LIN {X 0,Y 538.019,Z 685.461,A -85,B 0,C 180,E1 -4168.934,E2 -4168.934} C_VEL
LIN {X 0,Y 538.004,Z 685.465,A -85,B 0,C 180,E1 -4171.889,E2 -4171.889} C_VEL
LIN {X 0,Y 538.017,Z 685.462,A -85,B 0,C 180,E1 -4174.621,E2 -4174.621} C_VEL
LIN {X 0,Y 537.998,Z 685.467,A -85,B 0,C 180,E1 -4177.171,E2 -4177.171} C_VEL
LIN {X 0,Y 538.01,Z 685.465,A -85,B 0,C 180,E1 -4180.276,E2 -4180.276} C_VEL
LIN {X 0,Y 537.361,Z 685.545,A -85,B 0,C 180,E1 -4180.901,E2 -4180.901} C_VEL
LIN {X 0,Y 534.509,Z 685.908,A -85,B 0,C 180,E1 -4181.916,E2 -4181.916} C_VEL
LIN {X 0,Y 532.082,Z 686.21,A -85,B 0,C 180,E1 -4182.733,E2 -4182.733} C_VEL
LIN {X 0,Y 531.033,Z 686.336,A -85,B 0,C 180,E1 -4183.364,E2 -4183.364} C_VEL
LIN {X 0,Y 530.945,Z 686.346,A -85,B 0,C 180,E1 -4183.578,E2 -4183.578} C_VEL
LIN {X 0,Y 530.938,Z 686.345,A -85,B 0,C 180,E1 -4186.505,E2 -4186.505} C_VEL
LIN {X 0,Y 530.976,Z 686.345,A -85,B 0,C 180,E1 -4189.568,E2 -4189.568} C_VEL
LIN {X 0,Y 531.016,Z 686.543,A -85,B 0,C 180,E1 -4190.371,E2 -4190.371} C_VEL
LIN {X 0,Y 531.273,Z 687.633,A -85,B 0,C 180,E1 -4190.492,E2 -4190.492} C_VEL
LIN {X 0,Y 532.785,Z 692.095,A -85,B 0,C 180,E1 -4190.606,E2 -4190.606} C_VEL
LIN {X 0,Y 532.506,Z 766.443,A -85,B 0,C 180,E1 -4191.64,E2 -4191.64} C_VEL
LIN {X 0,Y 532.44,Z 779.405,A -85,B 0,C 180,E1 -4191.978,E2 -4191.978} C_VEL
LIN {X 0,Y 532.245,Z 791.35,A -85,B 0,C 180,E1 -4192.434,E2 -4192.434} C_VEL
LIN {X 0,Y 532.057,Z 803.366,A -85,B 0,C 180,E1 -4193.059,E2 -4193.059} C_VEL
LIN {X 0,Y 531.84,Z 814.43,A -85,B 0,C 180,E1 -4193.804,E2 -4193.804} C_VEL
LIN {X 0,Y 531.584,Z 824.165,A -85,B 0,C 180,E1 -4194.617,E2 -4194.617} C_VEL
LIN {X 0,Y 531.338,Z 833.433,A -85,B 0,C 180,E1 -4195.568,E2 -4195.568} C_VEL
LIN {X 0,Y 531.062,Z 842.493,A -85,B 0,C 180,E1 -4196.728,E2 -4196.728} C_VEL
LIN {X 0,Y 530.923,Z 849.848,A -85,B 0,C 180,E1 -4197.908,E2 -4197.908} C_VEL
LIN {X 0,Y 530.783,Z 856.177,A -85,B 0,C 180,E1 -4199.198,E2 -4199.198} C_VEL
LIN {X 0,Y 530.683,Z 860.138,A -85,B 0,C 180,E1 -4200.225,E2 -4200.225} C_VEL
LIN {X 0,Y 530.626,Z 863.895,A -85,B 0,C 180,E1 -4201.524,E2 -4201.524} C_VEL
LIN {X 0,Y 530.54,Z 866.036,A -85,B 0,C 180,E1 -4202.567,E2 -4202.567} C_VEL
LIN {X 0,Y 530.541,Z 866.991,A -85,B 0,C 180,E1 -4203.233,E2 -4203.233} C_VEL
LIN {X 0,Y 530.53,Z 867.86,A -85,B 0,C 180,E1 -4204.265,E2 -4204.265} C_VEL
LIN {X 0,Y 530.494,Z 867.898,A -85,B 0,C 180,E1 -4205.753,E2 -4205.753} C_VEL
LIN {X 0,Y 530.511,Z 867.253,A -85,B 0,C 180,E1 -4206.584,E2 -4206.584} C_VEL
LIN {X 0,Y 530.537,Z 865.086,A -85,B 0,C 180,E1 -4208.017,E2 -4208.017} C_VEL
LIN {X 0,Y 530.666,Z 861.391,A -85,B 0,C 180,E1 -4209.455,E2 -4209.455} C_VEL
LIN {X 0,Y 530.748,Z 857.026,A -85,B 0,C 180,E1 -4210.669,E2 -4210.669} C_VEL
LIN {X 0,Y 530.884,Z 851.4,A -85,B 0,C 180,E1 -4211.876,E2 -4211.876} C_VEL
LIN {X 0,Y 531.012,Z 844.363,A -85,B 0,C 180,E1 -4213.073,E2 -4213.073} C_VEL
LIN {X 0,Y 531.225,Z 837.108,A -85,B 0,C 180,E1 -4214.068,E2 -4214.068} C_VEL
LIN {X 0,Y 531.418,Z 828.24,A -85,B 0,C 180,E1 -4215.064,E2 -4215.064} C_VEL
LIN {X 0,Y 531.703,Z 817.426,A -85,B 0,C 180,E1 -4216.042,E2 -4216.042} C_VEL
LIN {X 0,Y 531.959,Z 806.49,A -85,B 0,C 180,E1 -4216.828,E2 -4216.828} C_VEL
LIN {X 0,Y 532.173,Z 795.377,A -85,B 0,C 180,E1 -4217.454,E2 -4217.454} C_VEL
LIN {X 0,Y 532.331,Z 783.475,A -85,B 0,C 180,E1 -4217.966,E2 -4217.966} C_VEL
LIN {X 0,Y 532.499,Z 770.64,A -85,B 0,C 180,E1 -4218.354,E2 -4218.354} C_VEL
LIN {X 0,Y 532.584,Z 756.116,A -85,B 0,C 180,E1 -4218.609,E2 -4218.609} C_VEL
LIN {X 0,Y 532.658,Z 691.597,A -85,B 0,C 180,E1 -4219.49,E2 -4219.49} C_VEL
LIN {X 0,Y 531.166,Z 687.265,A -85,B 0,C 180,E1 -4219.615,E2 -4219.615} C_VEL
LIN {X 0,Y 530.995,Z 686.43,A -85,B 0,C 180,E1 -4219.757,E2 -4219.757} C_VEL
LIN {X 0,Y 531.004,Z 686.341,A -85,B 0,C 180,E1 -4222.396,E2 -4222.396} C_VEL
LIN {X 0,Y 531.086,Z 686.328,A -85,B 0,C 180,E1 -4224.686,E2 -4224.686} C_VEL
LIN {X 0,Y 531.135,Z 686.324,A -85,B 0,C 180,E1 -4227.726,E2 -4227.726} C_VEL
LIN {X 0,Y 531.131,Z 686.327,A -85,B 0,C 180,E1 -4230.001,E2 -4230.001} C_VEL
LIN {X 0,Y 531.134,Z 686.327,A -85,B 0,C 180,E1 -4232.276,E2 -4232.276} C_VEL
LIN {X 0,Y 531.086,Z 686.326,A -85,B 0,C 180,E1 -4235.316,E2 -4235.316} C_VEL
LIN {X 0,Y 530.985,Z 686.344,A -85,B 0,C 180,E1 -4238.373,E2 -4238.373} C_VEL
LIN {X 0,Y 531.015,Z 686.333,A -85,B 0,C 180,E1 -4241.65,E2 -4241.65} C_VEL
LIN {X 0,Y 531.027,Z 686.337,A -85,B 0,C 180,E1 -4244.952,E2 -4244.952} C_VEL
LIN {X 0,Y 530.977,Z 686.338,A -85,B 0,C 180,E1 -4247.725,E2 -4247.725} C_VEL
LIN {X 0,Y 530.984,Z 686.344,A -85,B 0,C 180,E1 -4250.94,E2 -4250.94} C_VEL
LIN {X 0,Y 530.958,Z 686.341,A -85,B 0,C 180,E1 -4254.031,E2 -4254.031} C_VEL
LIN {X 0,Y 530.943,Z 686.343,A -85,B 0,C 180,E1 -4256.748,E2 -4256.748} C_VEL
LIN {X 0,Y 530.919,Z 686.353,A -85,B 0,C 180,E1 -4259.327,E2 -4259.327} C_VEL
LIN {X 0,Y 530.955,Z 686.34,A -85,B 0,C 180,E1 -4262.098,E2 -4262.098} C_VEL
LIN {X 0,Y 530.953,Z 686.338,A -85,B 0,C 180,E1 -4264.848,E2 -4264.848} C_VEL
LIN {X 0,Y 530.91,Z 686.354,A -85,B 0,C 180,E1 -4267.513,E2 -4267.513} C_VEL
LIN {X 0,Y 530.91,Z 686.346,A -85,B 0,C 180,E1 -4270.441,E2 -4270.441} C_VEL
LIN {X 0,Y 530.922,Z 686.354,A -85,B 0,C 180,E1 -4273.5,E2 -4273.5} C_VEL
LIN {X 0,Y 530.965,Z 686.35,A -85,B 0,C 180,E1 -4275.625,E2 -4275.625} C_VEL
LIN {X 0,Y 530.912,Z 686.347,A -85,B 0,C 180,E1 -4278.556,E2 -4278.556} C_VEL
LIN {X 0,Y 530.918,Z 686.351,A -85,B 0,C 180,E1 -4281.526,E2 -4281.526} C_VEL
LIN {X 0,Y 530.923,Z 686.349,A -85,B 0,C 180,E1 -4284.377,E2 -4284.377} C_VEL
LIN {X 0,Y 530.95,Z 686.343,A -85,B 0,C 180,E1 -4287.132,E2 -4287.132} C_VEL
LIN {X 0,Y 530.937,Z 686.352,A -85,B 0,C 180,E1 -4289.801,E2 -4289.801} C_VEL
LIN {X 0,Y 530.951,Z 686.525,A -85,B 0,C 180,E1 -4292.419,E2 -4292.419} C_VEL
LIN {X 0,Y 531.176,Z 687.511,A -85,B 0,C 180,E1 -4292.538,E2 -4292.538} C_VEL
LIN {X 0,Y 532.707,Z 692.815,A -85,B 0,C 180,E1 -4292.665,E2 -4292.665} C_VEL
LIN {X 0,Y 532.428,Z 761.148,A -85,B 0,C 180,E1 -4293.605,E2 -4293.605} C_VEL
LIN {X 0,Y 532.252,Z 773.625,A -85,B 0,C 180,E1 -4293.908,E2 -4293.908} C_VEL
LIN {X 0,Y 532.095,Z 783.825,A -85,B 0,C 180,E1 -4294.264,E2 -4294.264} C_VEL
LIN {X 0,Y 531.898,Z 792.983,A -85,B 0,C 180,E1 -4294.673,E2 -4294.673} C_VEL
LIN {X 0,Y 531.647,Z 803.731,A -85,B 0,C 180,E1 -4295.288,E2 -4295.288} C_VEL
LIN {X 0,Y 531.438,Z 813.803,A -85,B 0,C 180,E1 -4296.005,E2 -4296.005} C_VEL
LIN {X 0,Y 531.189,Z 822.13,A -85,B 0,C 180,E1 -4296.717,E2 -4296.717} C_VEL
LIN {X 0,Y 531.027,Z 830.575,A -85,B 0,C 180,E1 -4297.586,E2 -4297.586} C_VEL
LIN {X 0,Y 530.865,Z 837.62,A -85,B 0,C 180,E1 -4298.446,E2 -4298.446} C_VEL
LIN {X 0,Y 530.677,Z 844.505,A -85,B 0,C 180,E1 -4299.454,E2 -4299.454} C_VEL
LIN {X 0,Y 530.615,Z 849.821,A -85,B 0,C 180,E1 -4300.386,E2 -4300.386} C_VEL
LIN {X 0,Y 530.529,Z 854.839,A -85,B 0,C 180,E1 -4301.462,E2 -4301.462} C_VEL
LIN {X 0,Y 530.466,Z 858.836,A -85,B 0,C 180,E1 -4302.539,E2 -4302.539} C_VEL
LIN {X 0,Y 530.435,Z 861.509,A -85,B 0,C 180,E1 -4303.449,E2 -4303.449} C_VEL
LIN {X 0,Y 530.334,Z 863.99,A -85,B 0,C 180,E1 -4304.63,E2 -4304.63} C_VEL
LIN {X 0,Y 530.396,Z 865.686,A -85,B 0,C 180,E1 -4306.201,E2 -4306.201} C_VEL
LIN {X 0,Y 530.368,Z 865.993,A -85,B 0,C 180,E1 -4306.981,E2 -4306.981} C_VEL
LIN {X 0,Y 530.454,Z 865.042,A -85,B 0,C 180,E1 -4308.649,E2 -4308.649} C_VEL
LIN {X 0,Y 530.418,Z 864.223,A -85,B 0,C 180,E1 -4309.31,E2 -4309.31} C_VEL
LIN {X 0,Y 530.427,Z 860.91,A -85,B 0,C 180,E1 -4310.851,E2 -4310.851} C_VEL
LIN {X 0,Y 530.496,Z 857.268,A -85,B 0,C 180,E1 -4312.004,E2 -4312.004} C_VEL
LIN {X 0,Y 530.576,Z 852.512,A -85,B 0,C 180,E1 -4313.153,E2 -4313.153} C_VEL
LIN {X 0,Y 530.679,Z 847.651,A -85,B 0,C 180,E1 -4314.109,E2 -4314.109} C_VEL
LIN {X 0,Y 530.723,Z 841.822,A -85,B 0,C 180,E1 -4315.062,E2 -4315.062} C_VEL
LIN {X 0,Y 530.874,Z 834.803,A -85,B 0,C 180,E1 -4316.014,E2 -4316.014} C_VEL
LIN {X 0,Y 531.069,Z 826.32,A -85,B 0,C 180,E1 -4316.966,E2 -4316.966} C_VEL
LIN {X 0,Y 531.336,Z 817.064,A -85,B 0,C 180,E1 -4317.821,E2 -4317.821} C_VEL
LIN {X 0,Y 531.506,Z 808.475,A -85,B 0,C 180,E1 -4318.484,E2 -4318.484} C_VEL
LIN {X 0,Y 531.713,Z 799.665,A -85,B 0,C 180,E1 -4319.053,E2 -4319.053} C_VEL
LIN {X 0,Y 532.003,Z 788.626,A -85,B 0,C 180,E1 -4319.621,E2 -4319.621} C_VEL
LIN {X 0,Y 532.173,Z 777.264,A -85,B 0,C 180,E1 -4320.071,E2 -4320.071} C_VEL
LIN {X 0,Y 532.334,Z 766.23,A -85,B 0,C 180,E1 -4320.378,E2 -4320.378} C_VEL
LIN {X 0,Y 532.483,Z 752.801,A -85,B 0,C 180,E1 -4320.614,E2 -4320.614} C_VEL
LIN {X 0,Y 532.664,Z 691.69,A -85,B 0,C 180,E1 -4321.441,E2 -4321.441} C_VEL
LIN {X 0,Y 531.212,Z 687.28,A -85,B 0,C 180,E1 -4321.564,E2 -4321.564} C_VEL
LIN {X 0,Y 531.068,Z 686.399,A -85,B 0,C 180,E1 -4321.706,E2 -4321.706} C_VEL
LIN {X 0,Y 530.957,Z 686.35,A -85,B 0,C 180,E1 -4323.795,E2 -4323.795} C_VEL
LIN {X 0,Y 531.073,Z 686.336,A -85,B 0,C 180,E1 -4326.077,E2 -4326.077} C_VEL
LIN {X 0,Y 531.021,Z 686.335,A -85,B 0,C 180,E1 -4329.138,E2 -4329.138} C_VEL
LIN {X 0,Y 531.056,Z 686.332,A -85,B 0,C 180,E1 -4331.67,E2 -4331.67} C_VEL
LIN {X 0,Y 531.038,Z 686.333,A -85,B 0,C 180,E1 -4334.955,E2 -4334.955} C_VEL
LIN {X 0,Y 530.988,Z 686.339,A -85,B 0,C 180,E1 -4337.723,E2 -4337.723} C_VEL
LIN {X 0,Y 531.032,Z 686.337,A -85,B 0,C 180,E1 -4340.127,E2 -4340.127} C_VEL
LIN {X 0,Y 530.951,Z 686.351,A -85,B 0,C 180,E1 -4342.573,E2 -4342.573} C_VEL
LIN {X 0,Y 531.005,Z 686.34,A -85,B 0,C 180,E1 -4345.058,E2 -4345.058} C_VEL
LIN {X 0,Y 530.977,Z 686.34,A -85,B 0,C 180,E1 -4347.598,E2 -4347.598} C_VEL
LIN {X 0,Y 530.975,Z 686.341,A -85,B 0,C 180,E1 -4350.197,E2 -4350.197} C_VEL
LIN {X 0,Y 530.973,Z 686.348,A -85,B 0,C 180,E1 -4352.866,E2 -4352.866} C_VEL
LIN {X 0,Y 530.96,Z 686.343,A -85,B 0,C 180,E1 -4355.62,E2 -4355.62} C_VEL
LIN {X 0,Y 530.971,Z 686.343,A -85,B 0,C 180,E1 -4358.653,E2 -4358.653} C_VEL
LIN {X 0,Y 530.999,Z 686.343,A -85,B 0,C 180,E1 -4361.435,E2 -4361.435} C_VEL
LIN {X 0,Y 530.979,Z 686.34,A -85,B 0,C 180,E1 -4364.548,E2 -4364.548} C_VEL
LIN {X 0,Y 530.988,Z 686.341,A -85,B 0,C 180,E1 -4367.834,E2 -4367.834} C_VEL
LIN {X 0,Y 530.976,Z 686.339,A -85,B 0,C 180,E1 -4370.555,E2 -4370.555} C_VEL
LIN {X 0,Y 530.957,Z 686.349,A -85,B 0,C 180,E1 -4373.441,E2 -4373.441} C_VEL
LIN {X 0,Y 530.961,Z 686.345,A -85,B 0,C 180,E1 -4376.224,E2 -4376.224} C_VEL
LIN {X 0,Y 530.98,Z 686.346,A -85,B 0,C 180,E1 -4379.354,E2 -4379.354} C_VEL
LIN {X 0,Y 531.015,Z 686.517,A -85,B 0,C 180,E1 -4381.391,E2 -4381.391} C_VEL
LIN {X 0,Y 533.822,Z 698.543,A -85,B 0,C 180,E1 -4382.985,E2 -4382.985} C_VEL
LIN {X 0,Y 533.552,Z 714.425,A -85,B 0,C 180,E1 -4384.861,E2 -4384.861} C_VEL
LIN {X 0,Y 533.033,Z 740.726,A -85,B 0,C 180,E1 -4387.927,E2 -4387.927} C_VEL
LIN {X 0,Y 532.461,Z 766.852,A -85,B 0,C 180,E1 -4390.932,E2 -4390.932} C_VEL
LIN {X 0,Y 531.861,Z 792.067,A -85,B 0,C 180,E1 -4393.888,E2 -4393.888} C_VEL
LIN {X 0,Y 531.732,Z 802.117,A -85,B 0,C 180,E1 -4395.026,E2 -4395.026} C_VEL
LIN {X 0,Y 532.819,Z 811.338,A -85,B 0,C 180,E1 -4395.194,E2 -4395.194} C_VEL
LIN {X 0,Y 532.419,Z 911.896,A -85,B 0,C 180,E1 -4396.57,E2 -4396.57} C_VEL
LIN {X 0,Y 532.295,Z 924.422,A -85,B 0,C 180,E1 -4396.883,E2 -4396.883} C_VEL
LIN {X 0,Y 532.012,Z 937.345,A -85,B 0,C 180,E1 -4397.361,E2 -4397.361} C_VEL
LIN {X 0,Y 531.811,Z 949.29,A -85,B 0,C 180,E1 -4397.966,E2 -4397.966} C_VEL
LIN {X 0,Y 531.557,Z 961.181,A -85,B 0,C 180,E1 -4398.753,E2 -4398.753} C_VEL
LIN {X 0,Y 531.267,Z 971.593,A -85,B 0,C 180,E1 -4399.615,E2 -4399.615} C_VEL
LIN {X 0,Y 531.062,Z 980.092,A -85,B 0,C 180,E1 -4400.477,E2 -4400.477} C_VEL
LIN {X 0,Y 530.882,Z 987.952,A -85,B 0,C 180,E1 -4401.434,E2 -4401.434} C_VEL
LIN {X 0,Y 530.686,Z 995.615,A -85,B 0,C 180,E1 -4402.58,E2 -4402.58} C_VEL
LIN {X 0,Y 530.608,Z 1002.674,A -85,B 0,C 180,E1 -4403.916,E2 -4403.916} C_VEL
LIN {X 0,Y 530.459,Z 1007.369,A -85,B 0,C 180,E1 -4405.059,E2 -4405.059} C_VEL
LIN {X 0,Y 530.516,Z 1010.955,A -85,B 0,C 180,E1 -4406.201,E2 -4406.201} C_VEL
LIN {X 0,Y 530.457,Z 1012.805,A -85,B 0,C 180,E1 -4406.961,E2 -4406.961} C_VEL
LIN {X 0,Y 530.41,Z 1014.193,A -85,B 0,C 180,E1 -4407.721,E2 -4407.721} C_VEL
LIN {X 0,Y 530.344,Z 1015.785,A -85,B 0,C 180,E1 -4409.24,E2 -4409.24} C_VEL
LIN {X 0,Y 530.342,Z 1016,A -85,B 0,C 180,E1 -4409.999,E2 -4409.999} C_VEL
LIN {X 0,Y 530.36,Z 1015.186,A -85,B 0,C 180,E1 -4411.518,E2 -4411.518} C_VEL
LIN {X 0,Y 530.41,Z 1014.199,A -85,B 0,C 180,E1 -4412.277,E2 -4412.277} C_VEL
LIN {X 0,Y 530.456,Z 1012.812,A -85,B 0,C 180,E1 -4413.037,E2 -4413.037} C_VEL
LIN {X 0,Y 530.522,Z 1009.899,A -85,B 0,C 180,E1 -4414.177,E2 -4414.177} C_VEL
LIN {X 0,Y 530.524,Z 1005.953,A -85,B 0,C 180,E1 -4415.32,E2 -4415.32} C_VEL
LIN {X 0,Y 530.595,Z 1000.28,A -85,B 0,C 180,E1 -4416.579,E2 -4416.579} C_VEL
LIN {X 0,Y 530.756,Z 993.244,A -85,B 0,C 180,E1 -4417.799,E2 -4417.799} C_VEL
LIN {X 0,Y 530.926,Z 985.001,A -85,B 0,C 180,E1 -4418.947,E2 -4418.947} C_VEL
LIN {X 0,Y 531.138,Z 976.551,A -85,B 0,C 180,E1 -4419.904,E2 -4419.904} C_VEL
LIN {X 0,Y 531.411,Z 966.108,A -85,B 0,C 180,E1 -4420.862,E2 -4420.862} C_VEL
LIN {X 0,Y 531.701,Z 955.154,A -85,B 0,C 180,E1 -4421.669,E2 -4421.669} C_VEL
LIN {X 0,Y 531.932,Z 944.429,A -85,B 0,C 180,E1 -4422.3,E2 -4422.3} C_VEL
LIN {X 0,Y 532.107,Z 932.797,A -85,B 0,C 180,E1 -4422.829,E2 -4422.829} C_VEL
LIN {X 0,Y 532.326,Z 919.392,A -85,B 0,C 180,E1 -4423.26,E2 -4423.26} C_VEL
LIN {X 0,Y 532.49,Z 906.167,A -85,B 0,C 180,E1 -4423.523,E2 -4423.523} C_VEL
LIN {X 0,Y 532.747,Z 809.633,A -85,B 0,C 180,E1 -4424.832,E2 -4424.832} C_VEL
LIN {X 0,Y 531.693,Z 801.869,A -85,B 0,C 180,E1 -4424.988,E2 -4424.988} C_VEL
LIN {X 0,Y 532.257,Z 775.362,A -85,B 0,C 180,E1 -4428.066,E2 -4428.066} C_VEL
LIN {X 0,Y 532.768,Z 753.344,A -85,B 0,C 180,E1 -4430.622,E2 -4430.622} C_VEL
LIN {X 0,Y 533.187,Z 730.114,A -85,B 0,C 180,E1 -4433.292,E2 -4433.292} C_VEL
LIN {X 0,Y 533.697,Z 707.278,A -85,B 0,C 180,E1 -4435.94,E2 -4435.94} C_VEL
LIN {X 0,Y 533.702,Z 698.128,A -85,B 0,C 180,E1 -4437.019,E2 -4437.019} C_VEL
LIN {X 0,Y 531.054,Z 686.453,A -85,B 0,C 180,E1 -4438.58,E2 -4438.58} C_VEL
LIN {X 0,Y 530.962,Z 686.345,A -85,B 0,C 180,E1 -4441.967,E2 -4441.967} C_VEL
LIN {X 0,Y 530.965,Z 686.345,A -85,B 0,C 180,E1 -4444.85,E2 -4444.85} C_VEL
LIN {X 0,Y 530.959,Z 686.342,A -85,B 0,C 180,E1 -4447.506,E2 -4447.506} C_VEL
LIN {X 0,Y 530.974,Z 686.347,A -85,B 0,C 180,E1 -4450.432,E2 -4450.432} C_VEL
LIN {X 0,Y 530.957,Z 686.341,A -85,B 0,C 180,E1 -4453.493,E2 -4453.493} C_VEL
LIN {X 0,Y 530.96,Z 686.345,A -85,B 0,C 180,E1 -4456.505,E2 -4456.505} C_VEL
LIN {X 0,Y 530.976,Z 686.337,A -85,B 0,C 180,E1 -4459.567,E2 -4459.567} C_VEL
LIN {X 0,Y 530.96,Z 686.344,A -85,B 0,C 180,E1 -4462.576,E2 -4462.576} C_VEL
LIN {X 0,Y 530.992,Z 686.343,A -85,B 0,C 180,E1 -4465.31,E2 -4465.31} C_VEL
LIN {X 0,Y 530.961,Z 686.341,A -85,B 0,C 180,E1 -4468.031,E2 -4468.031} C_VEL
LIN {X 0,Y 530.997,Z 686.34,A -85,B 0,C 180,E1 -4470.87,E2 -4470.87} C_VEL
LIN {X 0,Y 531.001,Z 686.343,A -85,B 0,C 180,E1 -4473.256,E2 -4473.256} C_VEL
LIN {X 0,Y 530.986,Z 686.34,A -85,B 0,C 180,E1 -4475.957,E2 -4475.957} C_VEL
LIN {X 0,Y 530.988,Z 686.337,A -85,B 0,C 180,E1 -4479.062,E2 -4479.062} C_VEL
LIN {X 0,Y 531.005,Z 686.335,A -85,B 0,C 180,E1 -4482.277,E2 -4482.277} C_VEL
LIN {X 0,Y 531.007,Z 686.339,A -85,B 0,C 180,E1 -4485.436,E2 -4485.436} C_VEL
LIN {X 0,Y 531.024,Z 686.334,A -85,B 0,C 180,E1 -4488.55,E2 -4488.55} C_VEL
LIN {X 0,Y 531.045,Z 686.331,A -85,B 0,C 180,E1 -4491.629,E2 -4491.629} C_VEL
LIN {X 0,Y 531.111,Z 686.323,A -85,B 0,C 180,E1 -4494.685,E2 -4494.685} C_VEL
LIN {X 0,Y 531.124,Z 686.322,A -85,B 0,C 180,E1 -4497.725,E2 -4497.725} C_VEL
LIN {X 0,Y 531.144,Z 686.321,A -85,B 0,C 180,E1 -4500.758,E2 -4500.758} C_VEL
LIN {X 0,Y 531.097,Z 686.325,A -85,B 0,C 180,E1 -4503.034,E2 -4503.034} C_VEL
LIN {X 0,Y 531.063,Z 686.33,A -85,B 0,C 180,E1 -4506.077,E2 -4506.077} C_VEL
LIN {X 0,Y 531.046,Z 686.335,A -85,B 0,C 180,E1 -4508.371,E2 -4508.371} C_VEL
LIN {X 0,Y 531.047,Z 686.329,A -85,B 0,C 180,E1 -4511.676,E2 -4511.676} C_VEL
LIN {X 0,Y 531.019,Z 686.341,A -85,B 0,C 180,E1 -4514.956,E2 -4514.956} C_VEL
LIN {X 0,Y 530.969,Z 686.34,A -85,B 0,C 180,E1 -4517.724,E2 -4517.724} C_VEL
LIN {X 0,Y 531.013,Z 686.334,A -85,B 0,C 180,E1 -4520.128,E2 -4520.128} C_VEL
LIN {X 0,Y 530.934,Z 686.344,A -85,B 0,C 180,E1 -4522.574,E2 -4522.574} C_VEL
LIN {X 0,Y 530.963,Z 686.344,A -85,B 0,C 180,E1 -4525.06,E2 -4525.06} C_VEL
LIN {X 0,Y 531,Z 686.338,A -85,B 0,C 180,E1 -4527.597,E2 -4527.597} C_VEL
LIN {X 0,Y 530.964,Z 686.342,A -85,B 0,C 180,E1 -4530.646,E2 -4530.646} C_VEL
LIN {X 0,Y 530.98,Z 686.346,A -85,B 0,C 180,E1 -4533.774,E2 -4533.774} C_VEL
LIN {X 0,Y 530.957,Z 686.341,A -85,B 0,C 180,E1 -4536.559,E2 -4536.559} C_VEL
LIN {X 0,Y 530.971,Z 686.349,A -85,B 0,C 180,E1 -4539.855,E2 -4539.855} C_VEL
LIN {X 0,Y 530.973,Z 686.341,A -85,B 0,C 180,E1 -4542.458,E2 -4542.458} C_VEL
LIN {X 0,Y 530.945,Z 686.346,A -85,B 0,C 180,E1 -4543.578,E2 -4543.578} C_VEL
LIN {X 0,Y 530.271,Z 686.434,A -85,B 0,C 180,E1 -4544.211,E2 -4544.211} C_VEL
LIN {X 0,Y 527.416,Z 686.785,A -85,B 0,C 180,E1 -4545.24,E2 -4545.24} C_VEL
LIN {X 0,Y 525.008,Z 687.087,A -85,B 0,C 180,E1 -4546.069,E2 -4546.069} C_VEL
LIN {X 0,Y 523.976,Z 687.212,A -85,B 0,C 180,E1 -4546.708,E2 -4546.708} C_VEL
LIN {X 0,Y 523.893,Z 687.221,A -85,B 0,C 180,E1 -4546.925,E2 -4546.925} C_VEL
LIN {X 0,Y 523.943,Z 687.223,A -85,B 0,C 180,E1 -4549.922,E2 -4549.922} C_VEL
LIN {X 0,Y 524.013,Z 687.536,A -85,B 0,C 180,E1 -4550.197,E2 -4550.197} C_VEL
LIN {X 0,Y 524.354,Z 688.861,A -85,B 0,C 180,E1 -4550.302,E2 -4550.302} C_VEL
LIN {X 0,Y 525.99,Z 693.763,A -85,B 0,C 180,E1 -4550.425,E2 -4550.425} C_VEL
LIN {X 0,Y 525.643,Z 767.711,A -85,B 0,C 180,E1 -4551.468,E2 -4551.468} C_VEL
LIN {X 0,Y 525.588,Z 780.686,A -85,B 0,C 180,E1 -4551.815,E2 -4551.815} C_VEL
LIN {X 0,Y 525.406,Z 792.396,A -85,B 0,C 180,E1 -4552.27,E2 -4552.27} C_VEL
LIN {X 0,Y 525.214,Z 803.677,A -85,B 0,C 180,E1 -4552.857,E2 -4552.857} C_VEL
LIN {X 0,Y 524.989,Z 814.528,A -85,B 0,C 180,E1 -4553.585,E2 -4553.585} C_VEL
LIN {X 0,Y 524.696,Z 825.213,A -85,B 0,C 180,E1 -4554.482,E2 -4554.482} C_VEL
LIN {X 0,Y 524.411,Z 835.068,A -85,B 0,C 180,E1 -4555.515,E2 -4555.515} C_VEL
LIN {X 0,Y 524.127,Z 843.735,A -85,B 0,C 180,E1 -4556.651,E2 -4556.651} C_VEL
LIN {X 0,Y 523.944,Z 851.17,A -85,B 0,C 180,E1 -4557.867,E2 -4557.867} C_VEL
LIN {X 0,Y 523.793,Z 857.418,A -85,B 0,C 180,E1 -4559.174,E2 -4559.174} C_VEL
LIN {X 0,Y 523.675,Z 861.383,A -85,B 0,C 180,E1 -4560.229,E2 -4560.229} C_VEL
LIN {X 0,Y 523.606,Z 865.067,A -85,B 0,C 180,E1 -4561.545,E2 -4561.545} C_VEL
LIN {X 0,Y 523.512,Z 867.506,A -85,B 0,C 180,E1 -4562.844,E2 -4562.844} C_VEL
LIN {X 0,Y 523.497,Z 868.776,A -85,B 0,C 180,E1 -4564.091,E2 -4564.091} C_VEL
LIN {X 0,Y 523.476,Z 869.02,A -85,B 0,C 180,E1 -4565.407,E2 -4565.407} C_VEL
LIN {X 0,Y 523.492,Z 868.601,A -85,B 0,C 180,E1 -4566.251,E2 -4566.251} C_VEL
LIN {X 0,Y 523.492,Z 867.69,A -85,B 0,C 180,E1 -4567.089,E2 -4567.089} C_VEL
LIN {X 0,Y 523.511,Z 866.337,A -85,B 0,C 180,E1 -4567.922,E2 -4567.922} C_VEL
LIN {X 0,Y 523.677,Z 863.396,A -85,B 0,C 180,E1 -4569.169,E2 -4569.169} C_VEL
LIN {X 0,Y 523.735,Z 859.378,A -85,B 0,C 180,E1 -4570.4,E2 -4570.4} C_VEL
LIN {X 0,Y 523.851,Z 854.135,A -85,B 0,C 180,E1 -4571.624,E2 -4571.624} C_VEL
LIN {X 0,Y 524.008,Z 847.468,A -85,B 0,C 180,E1 -4572.84,E2 -4572.84} C_VEL
LIN {X 0,Y 524.261,Z 839.137,A -85,B 0,C 180,E1 -4574.05,E2 -4574.05} C_VEL
LIN {X 0,Y 524.493,Z 830.258,A -85,B 0,C 180,E1 -4575.09,E2 -4575.09} C_VEL
LIN {X 0,Y 524.767,Z 820.019,A -85,B 0,C 180,E1 -4576.052,E2 -4576.052} C_VEL
LIN {X 0,Y 525.06,Z 809.468,A -85,B 0,C 180,E1 -4576.849,E2 -4576.849} C_VEL
LIN {X 0,Y 525.296,Z 797.482,A -85,B 0,C 180,E1 -4577.561,E2 -4577.561} C_VEL
LIN {X 0,Y 525.463,Z 784.671,A -85,B 0,C 180,E1 -4578.128,E2 -4578.128} C_VEL
LIN {X 0,Y 525.628,Z 771.632,A -85,B 0,C 180,E1 -4578.529,E2 -4578.529} C_VEL
LIN {X 0,Y 525.713,Z 757.992,A -85,B 0,C 180,E1 -4578.775,E2 -4578.775} C_VEL
LIN {X 0,Y 525.902,Z 693.302,A -85,B 0,C 180,E1 -4579.668,E2 -4579.668} C_VEL
LIN {X 0,Y 524.121,Z 688.156,A -85,B 0,C 180,E1 -4579.816,E2 -4579.816} C_VEL
LIN {X 0,Y 523.946,Z 687.317,A -85,B 0,C 180,E1 -4579.959,E2 -4579.959} C_VEL
LIN {X 0,Y 523.995,Z 687.21,A -85,B 0,C 180,E1 -4583.068,E2 -4583.068} C_VEL
LIN {X 0,Y 523.951,Z 687.216,A -85,B 0,C 180,E1 -4585.385,E2 -4585.385} C_VEL
LIN {X 0,Y 524.106,Z 687.199,A -85,B 0,C 180,E1 -4587.696,E2 -4587.696} C_VEL
LIN {X 0,Y 524.099,Z 687.203,A -85,B 0,C 180,E1 -4590.001,E2 -4590.001} C_VEL
LIN {X 0,Y 524.105,Z 687.203,A -85,B 0,C 180,E1 -4592.307,E2 -4592.307} C_VEL
LIN {X 0,Y 524.007,Z 687.214,A -85,B 0,C 180,E1 -4596.161,E2 -4596.161} C_VEL
LIN {X 0,Y 523.945,Z 687.215,A -85,B 0,C 180,E1 -4599.264,E2 -4599.264} C_VEL
LIN {X 0,Y 523.926,Z 687.222,A -85,B 0,C 180,E1 -4602.395,E2 -4602.395} C_VEL
LIN {X 0,Y 523.922,Z 687.216,A -85,B 0,C 180,E1 -4605.563,E2 -4605.563} C_VEL
LIN {X 0,Y 523.916,Z 687.218,A -85,B 0,C 180,E1 -4607.972,E2 -4607.972} C_VEL
LIN {X 0,Y 523.935,Z 687.214,A -85,B 0,C 180,E1 -4610.413,E2 -4610.413} C_VEL
LIN {X 0,Y 523.911,Z 687.228,A -85,B 0,C 180,E1 -4612.895,E2 -4612.895} C_VEL
LIN {X 0,Y 523.87,Z 687.223,A -85,B 0,C 180,E1 -4615.424,E2 -4615.424} C_VEL
LIN {X 0,Y 523.902,Z 687.217,A -85,B 0,C 180,E1 -4618.004,E2 -4618.004} C_VEL
LIN {X 0,Y 523.903,Z 687.224,A -85,B 0,C 180,E1 -4620.846,E2 -4620.846} C_VEL
LIN {X 0,Y 523.914,Z 687.214,A -85,B 0,C 180,E1 -4623.726,E2 -4623.726} C_VEL
LIN {X 0,Y 523.862,Z 687.22,A -85,B 0,C 180,E1 -4626.394,E2 -4626.394} C_VEL
LIN {X 0,Y 523.89,Z 687.225,A -85,B 0,C 180,E1 -4629.089,E2 -4629.089} C_VEL
LIN {X 0,Y 523.88,Z 687.224,A -85,B 0,C 180,E1 -4632.127,E2 -4632.127} C_VEL
LIN {X 0,Y 523.934,Z 687.221,A -85,B 0,C 180,E1 -4635.312,E2 -4635.312} C_VEL
LIN {X 0,Y 523.881,Z 687.223,A -85,B 0,C 180,E1 -4638.7,E2 -4638.7} C_VEL
LIN {X 0,Y 523.89,Z 687.223,A -85,B 0,C 180,E1 -4641.086,E2 -4641.086} C_VEL
LIN {X 0,Y 523.846,Z 687.236,A -85,B 0,C 180,E1 -4643.821,E2 -4643.821} C_VEL
LIN {X 0,Y 523.902,Z 687.223,A -85,B 0,C 180,E1 -4646.632,E2 -4646.632} C_VEL
LIN {X 0,Y 523.913,Z 687.223,A -85,B 0,C 180,E1 -4649.353,E2 -4649.353} C_VEL
LIN {X 0,Y 523.919,Z 687.432,A -85,B 0,C 180,E1 -4652.236,E2 -4652.236} C_VEL
LIN {X 0,Y 524.149,Z 688.434,A -85,B 0,C 180,E1 -4652.351,E2 -4652.351} C_VEL
LIN {X 0,Y 525.775,Z 693.317,A -85,B 0,C 180,E1 -4652.478,E2 -4652.478} C_VEL
LIN {X 0,Y 525.513,Z 762.384,A -85,B 0,C 180,E1 -4653.448,E2 -4653.448} C_VEL
LIN {X 0,Y 525.351,Z 773.938,A -85,B 0,C 180,E1 -4653.73,E2 -4653.73} C_VEL
LIN {X 0,Y 525.193,Z 784.759,A -85,B 0,C 180,E1 -4654.114,E2 -4654.114} C_VEL
LIN {X 0,Y 524.97,Z 793.83,A -85,B 0,C 180,E1 -4654.528,E2 -4654.528} C_VEL
LIN {X 0,Y 524.719,Z 804.487,A -85,B 0,C 180,E1 -4655.151,E2 -4655.151} C_VEL
LIN {X 0,Y 524.479,Z 814.171,A -85,B 0,C 180,E1 -4655.854,E2 -4655.854} C_VEL
LIN {X 0,Y 524.214,Z 822.649,A -85,B 0,C 180,E1 -4656.598,E2 -4656.598} C_VEL
LIN {X 0,Y 524.063,Z 829.456,A -85,B 0,C 180,E1 -4657.299,E2 -4657.299} C_VEL
LIN {X 0,Y 523.842,Z 837.908,A -85,B 0,C 180,E1 -4658.349,E2 -4658.349} C_VEL
LIN {X 0,Y 523.606,Z 845.899,A -85,B 0,C 180,E1 -4659.575,E2 -4659.575} C_VEL
LIN {X 0,Y 523.5,Z 852.23,A -85,B 0,C 180,E1 -4660.797,E2 -4660.797} C_VEL
LIN {X 0,Y 523.419,Z 857.233,A -85,B 0,C 180,E1 -4662.011,E2 -4662.011} C_VEL
LIN {X 0,Y 523.347,Z 860.995,A -85,B 0,C 180,E1 -4663.218,E2 -4663.218} C_VEL
LIN {X 0,Y 523.246,Z 863.639,A -85,B 0,C 180,E1 -4664.417,E2 -4664.417} C_VEL
LIN {X 0,Y 523.282,Z 865.605,A -85,B 0,C 180,E1 -4666.01,E2 -4666.01} C_VEL
LIN {X 0,Y 523.266,Z 865.929,A -85,B 0,C 180,E1 -4666.801,E2 -4666.801} C_VEL
LIN {X 0,Y 523.321,Z 865.39,A -85,B 0,C 180,E1 -4668.378,E2 -4668.378} C_VEL
LIN {X 0,Y 523.347,Z 864.434,A -85,B 0,C 180,E1 -4669.163,E2 -4669.163} C_VEL
LIN {X 0,Y 523.32,Z 861.412,A -85,B 0,C 180,E1 -4670.726,E2 -4670.726} C_VEL
LIN {X 0,Y 523.401,Z 857.931,A -85,B 0,C 180,E1 -4671.895,E2 -4671.895} C_VEL
LIN {X 0,Y 523.494,Z 853.352,A -85,B 0,C 180,E1 -4673.06,E2 -4673.06} C_VEL
LIN {X 0,Y 523.607,Z 847.558,A -85,B 0,C 180,E1 -4674.222,E2 -4674.222} C_VEL
LIN {X 0,Y 523.737,Z 840.474,A -85,B 0,C 180,E1 -4675.382,E2 -4675.382} C_VEL
LIN {X 0,Y 523.891,Z 833.251,A -85,B 0,C 180,E1 -4676.346,E2 -4676.346} C_VEL
LIN {X 0,Y 524.092,Z 826.476,A -85,B 0,C 180,E1 -4677.117,E2 -4677.117} C_VEL
LIN {X 0,Y 524.343,Z 818.451,A -85,B 0,C 180,E1 -4677.887,E2 -4677.887} C_VEL
LIN {X 0,Y 524.584,Z 808.731,A -85,B 0,C 180,E1 -4678.656,E2 -4678.656} C_VEL
LIN {X 0,Y 524.821,Z 799.884,A -85,B 0,C 180,E1 -4679.233,E2 -4679.233} C_VEL
LIN {X 0,Y 525.099,Z 789.802,A -85,B 0,C 180,E1 -4679.76,E2 -4679.76} C_VEL
LIN {X 0,Y 525.292,Z 779.168,A -85,B 0,C 180,E1 -4680.192,E2 -4680.192} C_VEL
LIN {X 0,Y 525.419,Z 768.728,A -85,B 0,C 180,E1 -4680.503,E2 -4680.503} C_VEL
LIN {X 0,Y 525.581,Z 756.405,A -85,B 0,C 180,E1 -4680.742,E2 -4680.742} C_VEL
LIN {X 0,Y 525.757,Z 692.851,A -85,B 0,C 180,E1 -4681.62,E2 -4681.62} C_VEL
LIN {X 0,Y 524.204,Z 688.152,A -85,B 0,C 180,E1 -4681.753,E2 -4681.753} C_VEL
LIN {X 0,Y 524.069,Z 687.287,A -85,B 0,C 180,E1 -4681.897,E2 -4681.897} C_VEL
LIN {X 0,Y 523.912,Z 687.228,A -85,B 0,C 180,E1 -4683.846,E2 -4683.846} C_VEL
LIN {X 0,Y 524.031,Z 687.213,A -85,B 0,C 180,E1 -4686.159,E2 -4686.159} C_VEL
LIN {X 0,Y 523.991,Z 687.211,A -85,B 0,C 180,E1 -4689.262,E2 -4689.262} C_VEL
LIN {X 0,Y 524.006,Z 687.211,A -85,B 0,C 180,E1 -4691.737,E2 -4691.737} C_VEL
LIN {X 0,Y 524.001,Z 687.21,A -85,B 0,C 180,E1 -4695.052,E2 -4695.052} C_VEL
LIN {X 0,Y 523.954,Z 687.217,A -85,B 0,C 180,E1 -4697.969,E2 -4697.969} C_VEL
LIN {X 0,Y 523.979,Z 687.219,A -85,B 0,C 180,E1 -4700.41,E2 -4700.41} C_VEL
LIN {X 0,Y 523.917,Z 687.224,A -85,B 0,C 180,E1 -4702.893,E2 -4702.893} C_VEL
LIN {X 0,Y 523.941,Z 687.216,A -85,B 0,C 180,E1 -4705.419,E2 -4705.419} C_VEL
LIN {X 0,Y 523.924,Z 687.219,A -85,B 0,C 180,E1 -4708.002,E2 -4708.002} C_VEL
LIN {X 0,Y 523.951,Z 687.222,A -85,B 0,C 180,E1 -4710.854,E2 -4710.854} C_VEL
LIN {X 0,Y 523.936,Z 687.217,A -85,B 0,C 180,E1 -4713.729,E2 -4713.729} C_VEL
LIN {X 0,Y 523.909,Z 687.221,A -85,B 0,C 180,E1 -4716.401,E2 -4716.401} C_VEL
LIN {X 0,Y 523.925,Z 687.225,A -85,B 0,C 180,E1 -4719.084,E2 -4719.084} C_VEL
LIN {X 0,Y 523.958,Z 687.214,A -85,B 0,C 180,E1 -4722.119,E2 -4722.119} C_VEL
LIN {X 0,Y 523.948,Z 687.223,A -85,B 0,C 180,E1 -4725.31,E2 -4725.31} C_VEL
LIN {X 0,Y 523.962,Z 687.214,A -85,B 0,C 180,E1 -4728.689,E2 -4728.689} C_VEL
LIN {X 0,Y 523.919,Z 687.222,A -85,B 0,C 180,E1 -4731.897,E2 -4731.897} C_VEL
LIN {X 0,Y 523.928,Z 687.219,A -85,B 0,C 180,E1 -4734.911,E2 -4734.911} C_VEL
LIN {X 0,Y 523.941,Z 687.225,A -85,B 0,C 180,E1 -4737.679,E2 -4737.679} C_VEL
LIN {X 0,Y 523.959,Z 687.221,A -85,B 0,C 180,E1 -4740.676,E2 -4740.676} C_VEL
LIN {X 0,Y 524.001,Z 687.506,A -85,B 0,C 180,E1 -4741.203,E2 -4741.203} C_VEL
LIN {X 0,Y 526.786,Z 699.396,A -85,B 0,C 180,E1 -4742.809,E2 -4742.809} C_VEL
LIN {X 0,Y 526.928,Z 705.727,A -85,B 0,C 180,E1 -4743.58,E2 -4743.58} C_VEL
LIN {X 0,Y 526.241,Z 731.1,A -85,B 0,C 180,E1 -4746.589,E2 -4746.589} C_VEL
LIN {X 0,Y 525.804,Z 752.988,A -85,B 0,C 180,E1 -4749.157,E2 -4749.157} C_VEL
LIN {X 0,Y 525.196,Z 781.865,A -85,B 0,C 180,E1 -4752.476,E2 -4752.476} C_VEL
LIN {X 0,Y 524.785,Z 802.1,A -85,B 0,C 180,E1 -4754.822,E2 -4754.822} C_VEL
LIN {X 0,Y 525.958,Z 812.663,A -85,B 0,C 180,E1 -4755.014,E2 -4755.014} C_VEL
LIN {X 0,Y 525.522,Z 911.896,A -85,B 0,C 180,E1 -4756.39,E2 -4756.39} C_VEL
LIN {X 0,Y 525.382,Z 925.184,A -85,B 0,C 180,E1 -4756.731,E2 -4756.731} C_VEL
LIN {X 0,Y 525.101,Z 937.344,A -85,B 0,C 180,E1 -4757.192,E2 -4757.192} C_VEL
LIN {X 0,Y 524.87,Z 949.454,A -85,B 0,C 180,E1 -4757.815,E2 -4757.815} C_VEL
LIN {X 0,Y 524.573,Z 961.18,A -85,B 0,C 180,E1 -4758.601,E2 -4758.601} C_VEL
LIN {X 0,Y 524.269,Z 971.594,A -85,B 0,C 180,E1 -4759.475,E2 -4759.475} C_VEL
LIN {X 0,Y 524.056,Z 980.1,A -85,B 0,C 180,E1 -4760.349,E2 -4760.349} C_VEL
LIN {X 0,Y 523.848,Z 987.952,A -85,B 0,C 180,E1 -4761.318,E2 -4761.318} C_VEL
LIN {X 0,Y 523.634,Z 995.615,A -85,B 0,C 180,E1 -4762.48,E2 -4762.48} C_VEL
LIN {X 0,Y 523.519,Z 1002.674,A -85,B 0,C 180,E1 -4763.834,E2 -4763.834} C_VEL
LIN {X 0,Y 523.384,Z 1007.369,A -85,B 0,C 180,E1 -4764.992,E2 -4764.992} C_VEL
LIN {X 0,Y 523.443,Z 1010.955,A -85,B 0,C 180,E1 -4766.15,E2 -4766.15} C_VEL
LIN {X 0,Y 523.368,Z 1012.805,A -85,B 0,C 180,E1 -4766.92,E2 -4766.92} C_VEL
LIN {X 0,Y 523.334,Z 1014.193,A -85,B 0,C 180,E1 -4767.69,E2 -4767.69} C_VEL
LIN {X 0,Y 523.25,Z 1015.785,A -85,B 0,C 180,E1 -4769.229,E2 -4769.229} C_VEL
LIN {X 0,Y 523.246,Z 1016,A -85,B 0,C 180,E1 -4769.999,E2 -4769.999} C_VEL
LIN {X 0,Y 523.274,Z 1015.185,A -85,B 0,C 180,E1 -4771.538,E2 -4771.538} C_VEL
LIN {X 0,Y 523.334,Z 1014.198,A -85,B 0,C 180,E1 -4772.308,E2 -4772.308} C_VEL
LIN {X 0,Y 523.367,Z 1012.812,A -85,B 0,C 180,E1 -4773.078,E2 -4773.078} C_VEL
LIN {X 0,Y 523.441,Z 1009.899,A -85,B 0,C 180,E1 -4774.234,E2 -4774.234} C_VEL
LIN {X 0,Y 523.464,Z 1005.953,A -85,B 0,C 180,E1 -4775.392,E2 -4775.392} C_VEL
LIN {X 0,Y 523.52,Z 1000.742,A -85,B 0,C 180,E1 -4776.578,E2 -4776.578} C_VEL
LIN {X 0,Y 523.663,Z 994.474,A -85,B 0,C 180,E1 -4777.712,E2 -4777.712} C_VEL
LIN {X 0,Y 523.851,Z 986.487,A -85,B 0,C 180,E1 -4778.874,E2 -4778.874} C_VEL
LIN {X 0,Y 524.108,Z 978.345,A -85,B 0,C 180,E1 -4779.843,E2 -4779.843} C_VEL
LIN {X 0,Y 524.352,Z 968.411,A -85,B 0,C 180,E1 -4780.814,E2 -4780.814} C_VEL
LIN {X 0,Y 524.692,Z 957.102,A -85,B 0,C 180,E1 -4781.694,E2 -4781.694} C_VEL
LIN {X 0,Y 524.921,Z 946.194,A -85,B 0,C 180,E1 -4782.368,E2 -4782.368} C_VEL
LIN {X 0,Y 525.169,Z 934.002,A -85,B 0,C 180,E1 -4782.952,E2 -4782.952} C_VEL
LIN {X 0,Y 525.379,Z 921.221,A -85,B 0,C 180,E1 -4783.389,E2 -4783.389} C_VEL
LIN {X 0,Y 525.622,Z 907.677,A -85,B 0,C 180,E1 -4783.679,E2 -4783.679} C_VEL
LIN {X 0,Y 525.918,Z 810.49,A -85,B 0,C 180,E1 -4785.017,E2 -4785.017} C_VEL
LIN {X 0,Y 524.756,Z 801.853,A -85,B 0,C 180,E1 -4785.193,E2 -4785.193} C_VEL
LIN {X 0,Y 525.279,Z 777.023,A -85,B 0,C 180,E1 -4788.077,E2 -4788.077} C_VEL
LIN {X 0,Y 525.848,Z 750.19,A -85,B 0,C 180,E1 -4791.151,E2 -4791.151} C_VEL
LIN {X 0,Y 526.454,Z 723.9,A -85,B 0,C 180,E1 -4794.235,E2 -4794.235} C_VEL
LIN {X 0,Y 526.905,Z 700.783,A -85,B 0,C 180,E1 -4796.967,E2 -4796.967} C_VEL
LIN {X 0,Y 524.945,Z 691.706,A -85,B 0,C 180,E1 -4798.158,E2 -4798.158} C_VEL
LIN {X 0,Y 523.998,Z 687.341,A -85,B 0,C 180,E1 -4798.774,E2 -4798.774} C_VEL
LIN {X 0,Y 523.916,Z 687.221,A -85,B 0,C 180,E1 -4801.543,E2 -4801.543} C_VEL
LIN {X 0,Y 523.927,Z 687.221,A -85,B 0,C 180,E1 -4804.289,E2 -4804.289} C_VEL
LIN {X 0,Y 523.901,Z 687.223,A -85,B 0,C 180,E1 -4807.131,E2 -4807.131} C_VEL
LIN {X 0,Y 523.93,Z 687.221,A -85,B 0,C 180,E1 -4810.129,E2 -4810.129} C_VEL
LIN {X 0,Y 523.914,Z 687.221,A -85,B 0,C 180,E1 -4813.166,E2 -4813.166} C_VEL
LIN {X 0,Y 523.934,Z 687.215,A -85,B 0,C 180,E1 -4815.771,E2 -4815.771} C_VEL
LIN {X 0,Y 523.937,Z 687.223,A -85,B 0,C 180,E1 -4818.907,E2 -4818.907} C_VEL
LIN {X 0,Y 523.908,Z 687.219,A -85,B 0,C 180,E1 -4821.897,E2 -4821.897} C_VEL
LIN {X 0,Y 523.929,Z 687.219,A -85,B 0,C 180,E1 -4824.908,E2 -4824.908} C_VEL
LIN {X 0,Y 523.928,Z 687.219,A -85,B 0,C 180,E1 -4827.678,E2 -4827.678} C_VEL
LIN {X 0,Y 523.96,Z 687.214,A -85,B 0,C 180,E1 -4830.672,E2 -4830.672} C_VEL
LIN {X 0,Y 523.967,Z 687.216,A -85,B 0,C 180,E1 -4833.728,E2 -4833.728} C_VEL
LIN {X 0,Y 523.925,Z 687.218,A -85,B 0,C 180,E1 -4836.27,E2 -4836.27} C_VEL
LIN {X 0,Y 523.935,Z 687.214,A -85,B 0,C 180,E1 -4838.766,E2 -4838.766} C_VEL
LIN {X 0,Y 523.941,Z 687.218,A -85,B 0,C 180,E1 -4841.22,E2 -4841.22} C_VEL
LIN {X 0,Y 523.924,Z 687.223,A -85,B 0,C 180,E1 -4843.639,E2 -4843.639} C_VEL
LIN {X 0,Y 523.928,Z 687.221,A -85,B 0,C 180,E1 -4846.028,E2 -4846.028} C_VEL
LIN {X 0,Y 524,Z 687.211,A -85,B 0,C 180,E1 -4848.394,E2 -4848.394} C_VEL
LIN {X 0,Y 523.993,Z 687.208,A -85,B 0,C 180,E1 -4851.516,E2 -4851.516} C_VEL
LIN {X 0,Y 524.071,Z 687.2,A -85,B 0,C 180,E1 -4854.614,E2 -4854.614} C_VEL
LIN {X 0,Y 524.097,Z 687.197,A -85,B 0,C 180,E1 -4857.695,E2 -4857.695} C_VEL
LIN {X 0,Y 524.114,Z 687.197,A -85,B 0,C 180,E1 -4860.768,E2 -4860.768} C_VEL
LIN {X 0,Y 524.063,Z 687.201,A -85,B 0,C 180,E1 -4863.075,E2 -4863.075} C_VEL
LIN {X 0,Y 524.025,Z 687.207,A -85,B 0,C 180,E1 -4866.159,E2 -4866.159} C_VEL
LIN {X 0,Y 523.994,Z 687.215,A -85,B 0,C 180,E1 -4868.484,E2 -4868.484} C_VEL
LIN {X 0,Y 523.997,Z 687.207,A -85,B 0,C 180,E1 -4871.743,E2 -4871.743} C_VEL
LIN {X 0,Y 523.981,Z 687.216,A -85,B 0,C 180,E1 -4875.053,E2 -4875.053} C_VEL
LIN {X 0,Y 523.936,Z 687.216,A -85,B 0,C 180,E1 -4877.97,E2 -4877.97} C_VEL
LIN {X 0,Y 523.961,Z 687.213,A -85,B 0,C 180,E1 -4880.411,E2 -4880.411} C_VEL
LIN {X 0,Y 523.899,Z 687.224,A -85,B 0,C 180,E1 -4882.894,E2 -4882.894} C_VEL
LIN {X 0,Y 523.934,Z 687.218,A -85,B 0,C 180,E1 -4886.012,E2 -4886.012} C_VEL
LIN {X 0,Y 523.919,Z 687.217,A -85,B 0,C 180,E1 -4888.876,E2 -4888.876} C_VEL
LIN {X 0,Y 523.913,Z 687.226,A -85,B 0,C 180,E1 -4891.545,E2 -4891.545} C_VEL
LIN {X 0,Y 523.932,Z 687.218,A -85,B 0,C 180,E1 -4894.291,E2 -4894.291} C_VEL
LIN {X 0,Y 523.902,Z 687.222,A -85,B 0,C 180,E1 -4897.133,E2 -4897.133} C_VEL
LIN {X 0,Y 523.93,Z 687.222,A -85,B 0,C 180,E1 -4900.131,E2 -4900.131} C_VEL
LIN {X 0,Y 523.93,Z 687.219,A -85,B 0,C 180,E1 -4902.46,E2 -4902.46} C_VEL
LIN {X 0,Y 523.937,Z 687.219,A -85,B 0,C 180,E1 -4905.311,E2 -4905.311} C_VEL
LIN {X 0,Y 523.893,Z 687.221,A -85,B 0,C 180,E1 -4906.925,E2 -4906.925} C_VEL
LIN {X 0,Y 523.218,Z 687.308,A -85,B 0,C 180,E1 -4907.353,E2 -4907.353} C_VEL
LIN {X 0,Y 520.381,Z 687.668,A -85,B 0,C 180,E1 -4908.022,E2 -4908.022} C_VEL
LIN {X 0,Y 517.539,Z 688.016,A -85,B 0,C 180,E1 -4908.698,E2 -4908.698} C_VEL
LIN {X 0,Y 516.873,Z 688.098,A -85,B 0,C 180,E1 -4909.134,E2 -4909.134} C_VEL
LIN {X 0,Y 516.949,Z 688.312,A -85,B 0,C 180,E1 -4909.959,E2 -4909.959} C_VEL
LIN {X 0,Y 517.166,Z 689.311,A -85,B 0,C 180,E1 -4910.077,E2 -4910.077} C_VEL
LIN {X 0,Y 519.03,Z 694.702,A -85,B 0,C 180,E1 -4910.224,E2 -4910.224} C_VEL
LIN {X 0,Y 518.801,Z 768.631,A -85,B 0,C 180,E1 -4911.285,E2 -4911.285} C_VEL
LIN {X 0,Y 518.702,Z 782.085,A -85,B 0,C 180,E1 -4911.649,E2 -4911.649} C_VEL
LIN {X 0,Y 518.536,Z 793.844,A -85,B 0,C 180,E1 -4912.118,E2 -4912.118} C_VEL
LIN {X 0,Y 518.354,Z 805.165,A -85,B 0,C 180,E1 -4912.724,E2 -4912.724} C_VEL
LIN {X 0,Y 518.094,Z 816.139,A -85,B 0,C 180,E1 -4913.477,E2 -4913.477} C_VEL
LIN {X 0,Y 517.826,Z 825.767,A -85,B 0,C 180,E1 -4914.298,E2 -4914.298} C_VEL
LIN {X 0,Y 517.532,Z 834.707,A -85,B 0,C 180,E1 -4915.227,E2 -4915.227} C_VEL
LIN {X 0,Y 517.223,Z 843.691,A -85,B 0,C 180,E1 -4916.38,E2 -4916.38} C_VEL
LIN {X 0,Y 517.022,Z 850.341,A -85,B 0,C 180,E1 -4917.436,E2 -4917.436} C_VEL
LIN {X 0,Y 516.858,Z 856.563,A -85,B 0,C 180,E1 -4918.662,E2 -4918.662} C_VEL
LIN {X 0,Y 516.714,Z 861.091,A -85,B 0,C 180,E1 -4919.786,E2 -4919.786} C_VEL
LIN {X 0,Y 516.613,Z 865.175,A -85,B 0,C 180,E1 -4921.124,E2 -4921.124} C_VEL
LIN {X 0,Y 516.525,Z 867.966,A -85,B 0,C 180,E1 -4922.446,E2 -4922.446} C_VEL
LIN {X 0,Y 516.469,Z 869.691,A -85,B 0,C 180,E1 -4923.912,E2 -4923.912} C_VEL
LIN {X 0,Y 516.479,Z 870.094,A -85,B 0,C 180,E1 -4925.051,E2 -4925.051} C_VEL
LIN {X 0,Y 516.461,Z 869.83,A -85,B 0,C 180,E1 -4925.907,E2 -4925.907} C_VEL
LIN {X 0,Y 516.481,Z 869.126,A -85,B 0,C 180,E1 -4926.759,E2 -4926.759} C_VEL
LIN {X 0,Y 516.514,Z 867.794,A -85,B 0,C 180,E1 -4927.707,E2 -4927.707} C_VEL
LIN {X 0,Y 516.633,Z 865.336,A -85,B 0,C 180,E1 -4928.871,E2 -4928.871} C_VEL
LIN {X 0,Y 516.724,Z 861.612,A -85,B 0,C 180,E1 -4930.123,E2 -4930.123} C_VEL
LIN {X 0,Y 516.845,Z 856.701,A -85,B 0,C 180,E1 -4931.366,E2 -4931.366} C_VEL
LIN {X 0,Y 516.987,Z 850.475,A -85,B 0,C 180,E1 -4932.6,E2 -4932.6} C_VEL
LIN {X 0,Y 517.235,Z 842.673,A -85,B 0,C 180,E1 -4933.828,E2 -4933.828} C_VEL
LIN {X 0,Y 517.527,Z 833.917,A -85,B 0,C 180,E1 -4934.926,E2 -4934.926} C_VEL
LIN {X 0,Y 517.796,Z 823.734,A -85,B 0,C 180,E1 -4935.96,E2 -4935.96} C_VEL
LIN {X 0,Y 518.064,Z 813.863,A -85,B 0,C 180,E1 -4936.768,E2 -4936.768} C_VEL
LIN {X 0,Y 518.342,Z 802.895,A -85,B 0,C 180,E1 -4937.482,E2 -4937.482} C_VEL
LIN {X 0,Y 518.54,Z 790.429,A -85,B 0,C 180,E1 -4938.109,E2 -4938.109} C_VEL
LIN {X 0,Y 518.71,Z 777.678,A -85,B 0,C 180,E1 -4938.572,E2 -4938.572} C_VEL
LIN {X 0,Y 518.79,Z 764.759,A -85,B 0,C 180,E1 -4938.871,E2 -4938.871} C_VEL
LIN {X 0,Y 518.997,Z 694.58,A -85,B 0,C 180,E1 -4939.862,E2 -4939.862} C_VEL
LIN {X 0,Y 517.069,Z 689.051,A -85,B 0,C 180,E1 -4940.022,E2 -4940.022} C_VEL
LIN {X 0,Y 516.923,Z 688.191,A -85,B 0,C 180,E1 -4940.167,E2 -4940.167} C_VEL
LIN {X 0,Y 516.97,Z 688.085,A -85,B 0,C 180,E1 -4942.973,E2 -4942.973} C_VEL
LIN {X 0,Y 516.918,Z 688.092,A -85,B 0,C 180,E1 -4945.322,E2 -4945.322} C_VEL
LIN {X 0,Y 517.075,Z 688.075,A -85,B 0,C 180,E1 -4947.664,E2 -4947.664} C_VEL
LIN {X 0,Y 517.068,Z 688.078,A -85,B 0,C 180,E1 -4950.001,E2 -4950.001} C_VEL
LIN {X 0,Y 517.074,Z 688.079,A -85,B 0,C 180,E1 -4952.338,E2 -4952.338} C_VEL
LIN {X 0,Y 516.973,Z 688.091,A -85,B 0,C 180,E1 -4956.245,E2 -4956.245} C_VEL
LIN {X 0,Y 516.907,Z 688.092,A -85,B 0,C 180,E1 -4959.391,E2 -4959.391} C_VEL
LIN {X 0,Y 516.888,Z 688.102,A -85,B 0,C 180,E1 -4962.566,E2 -4962.566} C_VEL
LIN {X 0,Y 516.943,Z 688.088,A -85,B 0,C 180,E1 -4965.144,E2 -4965.144} C_VEL
LIN {X 0,Y 516.877,Z 688.097,A -85,B 0,C 180,E1 -4968.225,E2 -4968.225} C_VEL
LIN {X 0,Y 516.893,Z 688.095,A -85,B 0,C 180,E1 -4970.703,E2 -4970.703} C_VEL
LIN {X 0,Y 516.861,Z 688.102,A -85,B 0,C 180,E1 -4973.225,E2 -4973.225} C_VEL
LIN {X 0,Y 516.861,Z 688.092,A -85,B 0,C 180,E1 -4976.176,E2 -4976.176} C_VEL
LIN {X 0,Y 516.835,Z 688.098,A -85,B 0,C 180,E1 -4978.421,E2 -4978.421} C_VEL
LIN {X 0,Y 516.854,Z 688.107,A -85,B 0,C 180,E1 -4981.113,E2 -4981.113} C_VEL
LIN {X 0,Y 516.871,Z 688.089,A -85,B 0,C 180,E1 -4983.959,E2 -4983.959} C_VEL
LIN {X 0,Y 516.805,Z 688.1,A -85,B 0,C 180,E1 -4986.753,E2 -4986.753} C_VEL
LIN {X 0,Y 516.827,Z 688.107,A -85,B 0,C 180,E1 -4989.728,E2 -4989.728} C_VEL
LIN {X 0,Y 516.838,Z 688.101,A -85,B 0,C 180,E1 -4992.837,E2 -4992.837} C_VEL
LIN {X 0,Y 516.903,Z 688.093,A -85,B 0,C 180,E1 -4995.007,E2 -4995.007} C_VEL
LIN {X 0,Y 516.834,Z 688.102,A -85,B 0,C 180,E1 -4998.41,E2 -4998.41} C_VEL
LIN {X 0,Y 516.854,Z 688.101,A -85,B 0,C 180,E1 -5001.281,E2 -5001.281} C_VEL
LIN {X 0,Y 516.829,Z 688.103,A -85,B 0,C 180,E1 -5004.678,E2 -5004.678} C_VEL
LIN {X 0,Y 516.87,Z 688.1,A -85,B 0,C 180,E1 -5007.463,E2 -5007.463} C_VEL
LIN {X 0,Y 516.845,Z 688.108,A -85,B 0,C 180,E1 -5010.491,E2 -5010.491} C_VEL
LIN {X 0,Y 516.889,Z 688.294,A -85,B 0,C 180,E1 -5012.037,E2 -5012.037} C_VEL
LIN {X 0,Y 517.185,Z 689.552,A -85,B 0,C 180,E1 -5012.168,E2 -5012.168} C_VEL
LIN {X 0,Y 518.914,Z 694.686,A -85,B 0,C 180,E1 -5012.298,E2 -5012.298} C_VEL
LIN {X 0,Y 518.609,Z 762.969,A -85,B 0,C 180,E1 -5013.272,E2 -5013.272} C_VEL
LIN {X 0,Y 518.444,Z 775.394,A -85,B 0,C 180,E1 -5013.584,E2 -5013.584} C_VEL
LIN {X 0,Y 518.277,Z 785.763,A -85,B 0,C 180,E1 -5013.959,E2 -5013.959} C_VEL
LIN {X 0,Y 518.063,Z 794.828,A -85,B 0,C 180,E1 -5014.379,E2 -5014.379} C_VEL
LIN {X 0,Y 517.819,Z 805.487,A -85,B 0,C 180,E1 -5015.011,E2 -5015.011} C_VEL
LIN {X 0,Y 517.578,Z 814.753,A -85,B 0,C 180,E1 -5015.689,E2 -5015.689} C_VEL
LIN {X 0,Y 517.266,Z 823.644,A -85,B 0,C 180,E1 -5016.477,E2 -5016.477} C_VEL
LIN {X 0,Y 517.111,Z 830.99,A -85,B 0,C 180,E1 -5017.253,E2 -5017.253} C_VEL
LIN {X 0,Y 516.876,Z 838.863,A -85,B 0,C 180,E1 -5018.252,E2 -5018.252} C_VEL
LIN {X 0,Y 516.676,Z 844.424,A -85,B 0,C 180,E1 -5019.08,E2 -5019.08} C_VEL
LIN {X 0,Y 516.564,Z 850.188,A -85,B 0,C 180,E1 -5020.115,E2 -5020.115} C_VEL
LIN {X 0,Y 516.402,Z 855.671,A -85,B 0,C 180,E1 -5021.347,E2 -5021.347} C_VEL
LIN {X 0,Y 516.307,Z 859.888,A -85,B 0,C 180,E1 -5022.574,E2 -5022.574} C_VEL
LIN {X 0,Y 516.26,Z 862.159,A -85,B 0,C 180,E1 -5023.388,E2 -5023.388} C_VEL
LIN {X 0,Y 516.194,Z 865.043,A -85,B 0,C 180,E1 -5025.008,E2 -5025.008} C_VEL
LIN {X 0,Y 516.203,Z 865.969,A -85,B 0,C 180,E1 -5025.814,E2 -5025.814} C_VEL
LIN {X 0,Y 516.211,Z 866.345,A -85,B 0,C 180,E1 -5027.418,E2 -5027.418} C_VEL
LIN {X 0,Y 516.287,Z 865.67,A -85,B 0,C 180,E1 -5028.556,E2 -5028.556} C_VEL
LIN {X 0,Y 516.282,Z 864.021,A -85,B 0,C 180,E1 -5029.807,E2 -5029.807} C_VEL
LIN {X 0,Y 516.301,Z 861.409,A -85,B 0,C 180,E1 -5030.994,E2 -5030.994} C_VEL
LIN {X 0,Y 516.379,Z 857.833,A -85,B 0,C 180,E1 -5032.178,E2 -5032.178} C_VEL
LIN {X 0,Y 516.51,Z 853.124,A -85,B 0,C 180,E1 -5033.365,E2 -5033.365} C_VEL
LIN {X 0,Y 516.611,Z 848.368,A -85,B 0,C 180,E1 -5034.34,E2 -5034.34} C_VEL
LIN {X 0,Y 516.738,Z 842.605,A -85,B 0,C 180,E1 -5035.319,E2 -5035.319} C_VEL
LIN {X 0,Y 516.928,Z 835.651,A -85,B 0,C 180,E1 -5036.297,E2 -5036.297} C_VEL
LIN {X 0,Y 517.191,Z 827.205,A -85,B 0,C 180,E1 -5037.274,E2 -5037.274} C_VEL
LIN {X 0,Y 517.445,Z 819.108,A -85,B 0,C 180,E1 -5038.054,E2 -5038.054} C_VEL
LIN {X 0,Y 517.682,Z 810.676,A -85,B 0,C 180,E1 -5038.736,E2 -5038.736} C_VEL
LIN {X 0,Y 517.945,Z 800.314,A -85,B 0,C 180,E1 -5039.417,E2 -5039.417} C_VEL
LIN {X 0,Y 518.209,Z 790.059,A -85,B 0,C 180,E1 -5039.951,E2 -5039.951} C_VEL
LIN {X 0,Y 518.398,Z 779.863,A -85,B 0,C 180,E1 -5040.364,E2 -5040.364} C_VEL
LIN {X 0,Y 518.526,Z 769.231,A -85,B 0,C 180,E1 -5040.679,E2 -5040.679} C_VEL
LIN {X 0,Y 518.675,Z 756.546,A -85,B 0,C 180,E1 -5040.922,E2 -5040.922} C_VEL
LIN {X 0,Y 518.96,Z 694.522,A -85,B 0,C 180,E1 -5041.795,E2 -5041.795} C_VEL
LIN {X 0,Y 517.209,Z 689.036,A -85,B 0,C 180,E1 -5041.947,E2 -5041.947} C_VEL
LIN {X 0,Y 517.066,Z 688.171,A -85,B 0,C 180,E1 -5042.093,E2 -5042.093} C_VEL
LIN {X 0,Y 517.027,Z 688.082,A -85,B 0,C 180,E1 -5045.46,E2 -5045.46} C_VEL
LIN {X 0,Y 516.962,Z 688.09,A -85,B 0,C 180,E1 -5048.6,E2 -5048.6} C_VEL
LIN {X 0,Y 516.959,Z 688.09,A -85,B 0,C 180,E1 -5051.807,E2 -5051.807} C_VEL
LIN {X 0,Y 516.952,Z 688.087,A -85,B 0,C 180,E1 -5055.146,E2 -5055.146} C_VEL
LIN {X 0,Y 516.922,Z 688.096,A -85,B 0,C 180,E1 -5058.222,E2 -5058.222} C_VEL
LIN {X 0,Y 516.919,Z 688.098,A -85,B 0,C 180,E1 -5060.701,E2 -5060.701} C_VEL
LIN {X 0,Y 516.908,Z 688.093,A -85,B 0,C 180,E1 -5064.072,E2 -5064.072} C_VEL
LIN {X 0,Y 516.904,Z 688.1,A -85,B 0,C 180,E1 -5066.659,E2 -5066.659} C_VEL
LIN {X 0,Y 516.917,Z 688.092,A -85,B 0,C 180,E1 -5069.523,E2 -5069.523} C_VEL
LIN {X 0,Y 516.9,Z 688.097,A -85,B 0,C 180,E1 -5072.543,E2 -5072.543} C_VEL
LIN {X 0,Y 516.872,Z 688.101,A -85,B 0,C 180,E1 -5075.329,E2 -5075.329} C_VEL
LIN {X 0,Y 516.886,Z 688.095,A -85,B 0,C 180,E1 -5077.942,E2 -5077.942} C_VEL
LIN {X 0,Y 516.889,Z 688.098,A -85,B 0,C 180,E1 -5080.741,E2 -5080.741} C_VEL
LIN {X 0,Y 516.889,Z 688.098,A -85,B 0,C 180,E1 -5082.831,E2 -5082.831} C_VEL
LIN {X 0,Y 516.901,Z 688.098,A -85,B 0,C 180,E1 -5085.006,E2 -5085.006} C_VEL
LIN {X 0,Y 516.919,Z 688.09,A -85,B 0,C 180,E1 -5088.398,E2 -5088.398} C_VEL
LIN {X 0,Y 516.883,Z 688.1,A -85,B 0,C 180,E1 -5091.283,E2 -5091.283} C_VEL
LIN {X 0,Y 516.874,Z 688.099,A -85,B 0,C 180,E1 -5094.219,E2 -5094.219} C_VEL
LIN {X 0,Y 516.887,Z 688.098,A -85,B 0,C 180,E1 -5097.051,E2 -5097.051} C_VEL
LIN {X 0,Y 516.898,Z 688.102,A -85,B 0,C 180,E1 -5099.796,E2 -5099.796} C_VEL
LIN {X 0,Y 516.942,Z 688.316,A -85,B 0,C 180,E1 -5100.974,E2 -5100.974} C_VEL
LIN {X 0,Y 519.996,Z 701.609,A -85,B 0,C 180,E1 -5102.8,E2 -5102.8} C_VEL
LIN {X 0,Y 519.908,Z 710.897,A -85,B 0,C 180,E1 -5103.938,E2 -5103.938} C_VEL
LIN {X 0,Y 519.278,Z 733.729,A -85,B 0,C 180,E1 -5106.678,E2 -5106.678} C_VEL
LIN {X 0,Y 518.683,Z 758.167,A -85,B 0,C 180,E1 -5109.579,E2 -5109.579} C_VEL
LIN {X 0,Y 518.153,Z 782.691,A -85,B 0,C 180,E1 -5112.434,E2 -5112.434} C_VEL
LIN {X 0,Y 517.786,Z 801.678,A -85,B 0,C 180,E1 -5114.609,E2 -5114.609} C_VEL
LIN {X 0,Y 519.113,Z 812.051,A -85,B 0,C 180,E1 -5114.807,E2 -5114.807} C_VEL
LIN {X 0,Y 518.633,Z 911.896,A -85,B 0,C 180,E1 -5116.206,E2 -5116.206} C_VEL
LIN {X 0,Y 518.469,Z 925.183,A -85,B 0,C 180,E1 -5116.551,E2 -5116.551} C_VEL
LIN {X 0,Y 518.145,Z 938.465,A -85,B 0,C 180,E1 -5117.066,E2 -5117.066} C_VEL
LIN {X 0,Y 517.866,Z 950.61,A -85,B 0,C 180,E1 -5117.72,E2 -5117.72} C_VEL
LIN {X 0,Y 517.594,Z 962.47,A -85,B 0,C 180,E1 -5118.545,E2 -5118.545} C_VEL
LIN {X 0,Y 517.241,Z 972.635,A -85,B 0,C 180,E1 -5119.429,E2 -5119.429} C_VEL
LIN {X 0,Y 516.969,Z 981.776,A -85,B 0,C 180,E1 -5120.413,E2 -5120.413} C_VEL
LIN {X 0,Y 516.714,Z 990.68,A -85,B 0,C 180,E1 -5121.591,E2 -5121.591} C_VEL
LIN {X 0,Y 516.511,Z 997.842,A -85,B 0,C 180,E1 -5122.768,E2 -5122.768} C_VEL
LIN {X 0,Y 516.456,Z 1004.361,A -85,B 0,C 180,E1 -5124.141,E2 -5124.141} C_VEL
LIN {X 0,Y 516.271,Z 1008.673,A -85,B 0,C 180,E1 -5125.314,E2 -5125.314} C_VEL
LIN {X 0,Y 516.355,Z 1010.955,A -85,B 0,C 180,E1 -5126.097,E2 -5126.097} C_VEL
LIN {X 0,Y 516.282,Z 1012.804,A -85,B 0,C 180,E1 -5126.878,E2 -5126.878} C_VEL
LIN {X 0,Y 516.261,Z 1014.192,A -85,B 0,C 180,E1 -5127.658,E2 -5127.658} C_VEL
LIN {X 0,Y 516.16,Z 1015.785,A -85,B 0,C 180,E1 -5129.219,E2 -5129.219} C_VEL
LIN {X 0,Y 516.154,Z 1016,A -85,B 0,C 180,E1 -5129.999,E2 -5129.999} C_VEL
LIN {X 0,Y 516.191,Z 1015.185,A -85,B 0,C 180,E1 -5131.559,E2 -5131.559} C_VEL
LIN {X 0,Y 516.26,Z 1014.198,A -85,B 0,C 180,E1 -5132.339,E2 -5132.339} C_VEL
LIN {X 0,Y 516.282,Z 1012.812,A -85,B 0,C 180,E1 -5133.12,E2 -5133.12} C_VEL
LIN {X 0,Y 516.343,Z 1009.898,A -85,B 0,C 180,E1 -5134.292,E2 -5134.292} C_VEL
LIN {X 0,Y 516.405,Z 1005.952,A -85,B 0,C 180,E1 -5135.465,E2 -5135.465} C_VEL
LIN {X 0,Y 516.478,Z 1000.086,A -85,B 0,C 180,E1 -5136.797,E2 -5136.797} C_VEL
LIN {X 0,Y 516.639,Z 993.243,A -85,B 0,C 180,E1 -5138.014,E2 -5138.014} C_VEL
LIN {X 0,Y 516.865,Z 985.001,A -85,B 0,C 180,E1 -5139.192,E2 -5139.192} C_VEL
LIN {X 0,Y 517.095,Z 976.552,A -85,B 0,C 180,E1 -5140.176,E2 -5140.176} C_VEL
LIN {X 0,Y 517.44,Z 966.106,A -85,B 0,C 180,E1 -5141.159,E2 -5141.159} C_VEL
LIN {X 0,Y 517.755,Z 955.939,A -85,B 0,C 180,E1 -5141.933,E2 -5141.933} C_VEL
LIN {X 0,Y 518.045,Z 944.426,A -85,B 0,C 180,E1 -5142.635,E2 -5142.635} C_VEL
LIN {X 0,Y 518.279,Z 932.797,A -85,B 0,C 180,E1 -5143.177,E2 -5143.177} C_VEL
LIN {X 0,Y 518.535,Z 919.391,A -85,B 0,C 180,E1 -5143.619,E2 -5143.619} C_VEL
LIN {X 0,Y 518.727,Z 906.167,A -85,B 0,C 180,E1 -5143.889,E2 -5143.889} C_VEL
LIN {X 0,Y 519.069,Z 811.31,A -85,B 0,C 180,E1 -5145.204,E2 -5145.204} C_VEL
LIN {X 0,Y 517.782,Z 801.622,A -85,B 0,C 180,E1 -5145.393,E2 -5145.393} C_VEL
LIN {X 0,Y 518.25,Z 776.026,A -85,B 0,C 180,E1 -5148.328,E2 -5148.328} C_VEL
LIN {X 0,Y 518.907,Z 749.161,A -85,B 0,C 180,E1 -5151.448,E2 -5151.448} C_VEL
LIN {X 0,Y 519.56,Z 721.166,A -85,B 0,C 180,E1 -5154.791,E2 -5154.791} C_VEL
LIN {X 0,Y 520.001,Z 702.324,A -85,B 0,C 180,E1 -5157.053,E2 -5157.053} C_VEL
LIN {X 0,Y 517.095,Z 688.941,A -85,B 0,C 180,E1 -5158.847,E2 -5158.847} C_VEL
LIN {X 0,Y 516.942,Z 688.151,A -85,B 0,C 180,E1 -5159.023,E2 -5159.023} C_VEL
LIN {X 0,Y 516.869,Z 688.1,A -85,B 0,C 180,E1 -5162.024,E2 -5162.024} C_VEL
LIN {X 0,Y 516.878,Z 688.101,A -85,B 0,C 180,E1 -5164.824,E2 -5164.824} C_VEL
LIN {X 0,Y 516.874,Z 688.099,A -85,B 0,C 180,E1 -5167.942,E2 -5167.942} C_VEL
LIN {X 0,Y 516.876,Z 688.103,A -85,B 0,C 180,E1 -5170.741,E2 -5170.741} C_VEL
LIN {X 0,Y 516.876,Z 688.101,A -85,B 0,C 180,E1 -5172.83,E2 -5172.83} C_VEL
LIN {X 0,Y 516.915,Z 688.095,A -85,B 0,C 180,E1 -5175.009,E2 -5175.009} C_VEL
LIN {X 0,Y 516.909,Z 688.095,A -85,B 0,C 180,E1 -5178.397,E2 -5178.397} C_VEL
LIN {X 0,Y 516.875,Z 688.101,A -85,B 0,C 180,E1 -5181.283,E2 -5181.283} C_VEL
LIN {X 0,Y 516.882,Z 688.091,A -85,B 0,C 180,E1 -5184.22,E2 -5184.22} C_VEL
LIN {X 0,Y 516.886,Z 688.101,A -85,B 0,C 180,E1 -5187.052,E2 -5187.052} C_VEL
LIN {X 0,Y 516.891,Z 688.096,A -85,B 0,C 180,E1 -5189.796,E2 -5189.796} C_VEL
LIN {X 0,Y 516.92,Z 688.089,A -85,B 0,C 180,E1 -5192.467,E2 -5192.467} C_VEL
LIN {X 0,Y 516.901,Z 688.095,A -85,B 0,C 180,E1 -5195.071,E2 -5195.071} C_VEL
LIN {X 0,Y 516.874,Z 688.093,A -85,B 0,C 180,E1 -5198.462,E2 -5198.462} C_VEL
LIN {X 0,Y 516.892,Z 688.094,A -85,B 0,C 180,E1 -5200.954,E2 -5200.954} C_VEL
LIN {X 0,Y 516.901,Z 688.094,A -85,B 0,C 180,E1 -5203.41,E2 -5203.41} C_VEL
LIN {X 0,Y 516.883,Z 688.102,A -85,B 0,C 180,E1 -5205.833,E2 -5205.833} C_VEL
LIN {X 0,Y 516.953,Z 688.091,A -85,B 0,C 180,E1 -5208.233,E2 -5208.233} C_VEL
LIN {X 0,Y 516.957,Z 688.083,A -85,B 0,C 180,E1 -5211.4,E2 -5211.4} C_VEL
LIN {X 0,Y 516.991,Z 688.085,A -85,B 0,C 180,E1 -5213.757,E2 -5213.757} C_VEL
LIN {X 0,Y 517.004,Z 688.08,A -85,B 0,C 180,E1 -5216.883,E2 -5216.883} C_VEL
LIN {X 0,Y 517.07,Z 688.074,A -85,B 0,C 180,E1 -5220,E2 -5220} C_VEL
LIN {X 0,Y 517.004,Z 688.08,A -85,B 0,C 180,E1 -5223.117,E2 -5223.117} C_VEL
LIN {X 0,Y 516.99,Z 688.085,A -85,B 0,C 180,E1 -5226.244,E2 -5226.244} C_VEL
LIN {X 0,Y 516.944,Z 688.087,A -85,B 0,C 180,E1 -5229.39,E2 -5229.39} C_VEL
LIN {X 0,Y 516.945,Z 688.086,A -85,B 0,C 180,E1 -5231.811,E2 -5231.811} C_VEL
LIN {X 0,Y 516.932,Z 688.092,A -85,B 0,C 180,E1 -5235.147,E2 -5235.147} C_VEL
LIN {X 0,Y 516.905,Z 688.092,A -85,B 0,C 180,E1 -5238.223,E2 -5238.223} C_VEL
LIN {X 0,Y 516.901,Z 688.096,A -85,B 0,C 180,E1 -5240.702,E2 -5240.702} C_VEL
LIN {X 0,Y 516.876,Z 688.092,A -85,B 0,C 180,E1 -5244.074,E2 -5244.074} C_VEL
LIN {X 0,Y 516.898,Z 688.095,A -85,B 0,C 180,E1 -5246.66,E2 -5246.66} C_VEL
LIN {X 0,Y 516.9,Z 688.1,A -85,B 0,C 180,E1 -5249.525,E2 -5249.525} C_VEL
LIN {X 0,Y 516.888,Z 688.091,A -85,B 0,C 180,E1 -5252.545,E2 -5252.545} C_VEL
LIN {X 0,Y 516.87,Z 688.102,A -85,B 0,C 180,E1 -5255.333,E2 -5255.333} C_VEL
LIN {X 0,Y 516.872,Z 688.1,A -85,B 0,C 180,E1 -5257.944,E2 -5257.944} C_VEL
LIN {X 0,Y 516.877,Z 688.096,A -85,B 0,C 180,E1 -5260.743,E2 -5260.743} C_VEL
LIN {X 0,Y 516.876,Z 688.096,A -85,B 0,C 180,E1 -5262.833,E2 -5262.833} C_VEL
LIN {X 0,Y 516.888,Z 688.096,A -85,B 0,C 180,E1 -5265.008,E2 -5265.008} C_VEL
LIN {X 0,Y 516.904,Z 688.096,A -85,B 0,C 180,E1 -5268.401,E2 -5268.401} C_VEL
LIN {X 0,Y 516.873,Z 688.098,A -85,B 0,C 180,E1 -5269.134,E2 -5269.134} C_VEL
LIN {X 0,Y 516.732,Z 688.777,A -85,B 0,C 180,E1 -5269.414,E2 -5269.414} C_VEL
LIN {X 0,Y 516.261,Z 691.037,A -85,B 0,C 180,E1 -5269.719,E2 -5269.719} C_VEL
LIN {X 0,Y 515.429,Z 695.096,A -85,B 0,C 180,E1 -5269.988,E2 -5269.988} C_VEL
LIN {X 0,Y 514.491,Z 699.894,A -85,B 0,C 180,E1 -5270.138,E2 -5270.138} C_VEL
LIN {X 0,Y 512.959,Z 707.919,A -85,B 0,C 180,E1 -5270.221,E2 -5270.221} C_VEL
LIN {X 0,Y 512.205,Z 717.211,A -85,B 0,C 180,E1 -5270.331,E2 -5270.331} C_VEL
LIN {X 0,Y 511.972,Z 769.23,A -85,B 0,C 180,E1 -5271.09,E2 -5271.09} C_VEL
LIN {X 0,Y 511.891,Z 781.779,A -85,B 0,C 180,E1 -5271.425,E2 -5271.425} C_VEL
LIN {X 0,Y 511.702,Z 793.687,A -85,B 0,C 180,E1 -5271.89,E2 -5271.89} C_VEL
LIN {X 0,Y 511.494,Z 805.186,A -85,B 0,C 180,E1 -5272.495,E2 -5272.495} C_VEL
LIN {X 0,Y 511.234,Z 816.586,A -85,B 0,C 180,E1 -5273.275,E2 -5273.275} C_VEL
LIN {X 0,Y 510.921,Z 827.294,A -85,B 0,C 180,E1 -5274.2,E2 -5274.2} C_VEL
LIN {X 0,Y 510.608,Z 836.375,A -85,B 0,C 180,E1 -5275.167,E2 -5275.167} C_VEL
LIN {X 0,Y 510.326,Z 843.598,A -85,B 0,C 180,E1 -5276.101,E2 -5276.101} C_VEL
LIN {X 0,Y 510.12,Z 850.527,A -85,B 0,C 180,E1 -5277.184,E2 -5277.184} C_VEL
LIN {X 0,Y 509.908,Z 856.885,A -85,B 0,C 180,E1 -5278.418,E2 -5278.418} C_VEL
LIN {X 0,Y 509.712,Z 862.355,A -85,B 0,C 180,E1 -5279.785,E2 -5279.785} C_VEL
LIN {X 0,Y 509.613,Z 866.374,A -85,B 0,C 180,E1 -5281.141,E2 -5281.141} C_VEL
LIN {X 0,Y 509.548,Z 868.317,A -85,B 0,C 180,E1 -5282.035,E2 -5282.035} C_VEL
LIN {X 0,Y 509.494,Z 869.721,A -85,B 0,C 180,E1 -5282.923,E2 -5282.923} C_VEL
LIN {X 0,Y 509.45,Z 870.648,A -85,B 0,C 180,E1 -5283.805,E2 -5283.805} C_VEL
LIN {X 0,Y 509.462,Z 871.043,A -85,B 0,C 180,E1 -5284.683,E2 -5284.683} C_VEL
LIN {X 0,Y 509.428,Z 871,A -85,B 0,C 180,E1 -5285.579,E2 -5285.579} C_VEL
LIN {X 0,Y 509.455,Z 870.493,A -85,B 0,C 180,E1 -5286.42,E2 -5286.42} C_VEL
LIN {X 0,Y 509.493,Z 869.127,A -85,B 0,C 180,E1 -5287.55,E2 -5287.55} C_VEL
LIN {X 0,Y 509.638,Z 866.156,A -85,B 0,C 180,E1 -5288.991,E2 -5288.991} C_VEL
LIN {X 0,Y 509.726,Z 862.376,A -85,B 0,C 180,E1 -5290.258,E2 -5290.258} C_VEL
LIN {X 0,Y 509.871,Z 857.396,A -85,B 0,C 180,E1 -5291.518,E2 -5291.518} C_VEL
LIN {X 0,Y 510.032,Z 851.101,A -85,B 0,C 180,E1 -5292.768,E2 -5292.768} C_VEL
LIN {X 0,Y 510.329,Z 843.166,A -85,B 0,C 180,E1 -5294.014,E2 -5294.014} C_VEL
LIN {X 0,Y 510.602,Z 835.028,A -85,B 0,C 180,E1 -5295.045,E2 -5295.045} C_VEL
LIN {X 0,Y 510.889,Z 825.103,A -85,B 0,C 180,E1 -5296.071,E2 -5296.071} C_VEL
LIN {X 0,Y 511.16,Z 815.333,A -85,B 0,C 180,E1 -5296.889,E2 -5296.889} C_VEL
LIN {X 0,Y 511.482,Z 803.373,A -85,B 0,C 180,E1 -5297.679,E2 -5297.679} C_VEL
LIN {X 0,Y 511.71,Z 790.778,A -85,B 0,C 180,E1 -5298.313,E2 -5298.313} C_VEL
LIN {X 0,Y 511.867,Z 778.164,A -85,B 0,C 180,E1 -5298.768,E2 -5298.768} C_VEL
LIN {X 0,Y 511.927,Z 765.014,A -85,B 0,C 180,E1 -5299.07,E2 -5299.07} C_VEL
LIN {X 0,Y 512.243,Z 696.209,A -85,B 0,C 180,E1 -5300.051,E2 -5300.051} C_VEL
LIN {X 0,Y 510.048,Z 689.924,A -85,B 0,C 180,E1 -5300.234,E2 -5300.234} C_VEL
LIN {X 0,Y 509.891,Z 689.068,A -85,B 0,C 180,E1 -5300.381,E2 -5300.381} C_VEL
LIN {X 0,Y 509.925,Z 688.964,A -85,B 0,C 180,E1 -5303.671,E2 -5303.671} C_VEL
LIN {X 0,Y 509.887,Z 688.969,A -85,B 0,C 180,E1 -5306.841,E2 -5306.841} C_VEL
LIN {X 0,Y 509.926,Z 688.969,A -85,B 0,C 180,E1 -5308.422,E2 -5308.422} C_VEL
LIN {X 0,Y 510.037,Z 688.954,A -85,B 0,C 180,E1 -5310.001,E2 -5310.001} C_VEL
LIN {X 0,Y 510.043,Z 688.955,A -85,B 0,C 180,E1 -5312.37,E2 -5312.37} C_VEL
LIN {X 0,Y 509.94,Z 688.961,A -85,B 0,C 180,E1 -5315.537,E2 -5315.537} C_VEL
LIN {X 0,Y 509.879,Z 688.967,A -85,B 0,C 180,E1 -5317.924,E2 -5317.924} C_VEL
LIN {X 0,Y 509.861,Z 688.971,A -85,B 0,C 180,E1 -5321.128,E2 -5321.128} C_VEL
LIN {X 0,Y 509.852,Z 688.974,A -85,B 0,C 180,E1 -5324.367,E2 -5324.367} C_VEL
LIN {X 0,Y 509.851,Z 688.979,A -85,B 0,C 180,E1 -5326.827,E2 -5326.827} C_VEL
LIN {X 0,Y 509.852,Z 688.966,A -85,B 0,C 180,E1 -5330.159,E2 -5330.159} C_VEL
LIN {X 0,Y 509.825,Z 688.979,A -85,B 0,C 180,E1 -5332.706,E2 -5332.706} C_VEL
LIN {X 0,Y 509.784,Z 688.978,A -85,B 0,C 180,E1 -5335.302,E2 -5335.302} C_VEL
LIN {X 0,Y 509.813,Z 688.972,A -85,B 0,C 180,E1 -5338.082,E2 -5338.082} C_VEL
LIN {X 0,Y 509.821,Z 688.981,A -85,B 0,C 180,E1 -5341.274,E2 -5341.274} C_VEL
LIN {X 0,Y 509.825,Z 688.965,A -85,B 0,C 180,E1 -5344.417,E2 -5344.417} C_VEL
LIN {X 0,Y 509.768,Z 688.984,A -85,B 0,C 180,E1 -5347.346,E2 -5347.346} C_VEL
LIN {X 0,Y 509.791,Z 688.978,A -85,B 0,C 180,E1 -5350.388,E2 -5350.388} C_VEL
LIN {X 0,Y 509.796,Z 688.987,A -85,B 0,C 180,E1 -5353.576,E2 -5353.576} C_VEL
LIN {X 0,Y 509.797,Z 688.978,A -85,B 0,C 180,E1 -5356.425,E2 -5356.425} C_VEL
LIN {X 0,Y 509.792,Z 688.985,A -85,B 0,C 180,E1 -5359.613,E2 -5359.613} C_VEL
LIN {X 0,Y 509.755,Z 688.983,A -85,B 0,C 180,E1 -5362.653,E2 -5362.653} C_VEL
LIN {X 0,Y 509.834,Z 688.981,A -85,B 0,C 180,E1 -5365.803,E2 -5365.803} C_VEL
LIN {X 0,Y 509.821,Z 688.979,A -85,B 0,C 180,E1 -5368.726,E2 -5368.726} C_VEL
LIN {X 0,Y 509.821,Z 689.173,A -85,B 0,C 180,E1 -5371.833,E2 -5371.833} C_VEL
LIN {X 0,Y 510.094,Z 690.292,A -85,B 0,C 180,E1 -5371.962,E2 -5371.962} C_VEL
LIN {X 0,Y 512.12,Z 696.28,A -85,B 0,C 180,E1 -5372.118,E2 -5372.118} C_VEL
LIN {X 0,Y 511.699,Z 764.372,A -85,B 0,C 180,E1 -5373.111,E2 -5373.111} C_VEL
LIN {X 0,Y 511.562,Z 776.179,A -85,B 0,C 180,E1 -5373.412,E2 -5373.412} C_VEL
LIN {X 0,Y 511.369,Z 787.152,A -85,B 0,C 180,E1 -5373.817,E2 -5373.817} C_VEL
LIN {X 0,Y 511.161,Z 795.826,A -85,B 0,C 180,E1 -5374.226,E2 -5374.226} C_VEL
LIN {X 0,Y 510.91,Z 806.059,A -85,B 0,C 180,E1 -5374.837,E2 -5374.837} C_VEL
LIN {X 0,Y 510.679,Z 815.037,A -85,B 0,C 180,E1 -5375.494,E2 -5375.494} C_VEL
LIN {X 0,Y 510.376,Z 823.608,A -85,B 0,C 180,E1 -5376.248,E2 -5376.248} C_VEL
LIN {X 0,Y 510.179,Z 831.645,A -85,B 0,C 180,E1 -5377.097,E2 -5377.097} C_VEL
LIN {X 0,Y 509.966,Z 838.552,A -85,B 0,C 180,E1 -5377.959,E2 -5377.959} C_VEL
LIN {X 0,Y 509.694,Z 845.435,A -85,B 0,C 180,E1 -5378.991,E2 -5378.991} C_VEL
LIN {X 0,Y 509.587,Z 850.177,A -85,B 0,C 180,E1 -5379.831,E2 -5379.831} C_VEL
LIN {X 0,Y 509.446,Z 855.931,A -85,B 0,C 180,E1 -5381.083,E2 -5381.083} C_VEL
LIN {X 0,Y 509.324,Z 860.339,A -85,B 0,C 180,E1 -5382.328,E2 -5382.328} C_VEL
LIN {X 0,Y 509.262,Z 862.647,A -85,B 0,C 180,E1 -5383.153,E2 -5383.153} C_VEL
LIN {X 0,Y 509.2,Z 865.832,A -85,B 0,C 180,E1 -5384.797,E2 -5384.797} C_VEL
LIN {X 0,Y 509.194,Z 866.792,A -85,B 0,C 180,E1 -5385.615,E2 -5385.615} C_VEL
LIN {X 0,Y 509.198,Z 867.456,A -85,B 0,C 180,E1 -5387.242,E2 -5387.242} C_VEL
LIN {X 0,Y 509.267,Z 866.824,A -85,B 0,C 180,E1 -5388.473,E2 -5388.473} C_VEL
LIN {X 0,Y 509.266,Z 865.37,A -85,B 0,C 180,E1 -5389.665,E2 -5389.665} C_VEL
LIN {X 0,Y 509.273,Z 862.941,A -85,B 0,C 180,E1 -5390.868,E2 -5390.868} C_VEL
LIN {X 0,Y 509.377,Z 859.511,A -85,B 0,C 180,E1 -5392.069,E2 -5392.069} C_VEL
LIN {X 0,Y 509.526,Z 854.941,A -85,B 0,C 180,E1 -5393.277,E2 -5393.277} C_VEL
LIN {X 0,Y 509.632,Z 849.261,A -85,B 0,C 180,E1 -5394.46,E2 -5394.46} C_VEL
LIN {X 0,Y 509.803,Z 843.446,A -85,B 0,C 180,E1 -5395.453,E2 -5395.453} C_VEL
LIN {X 0,Y 509.998,Z 836.446,A -85,B 0,C 180,E1 -5396.445,E2 -5396.445} C_VEL
LIN {X 0,Y 510.288,Z 827.936,A -85,B 0,C 180,E1 -5397.434,E2 -5397.434} C_VEL
LIN {X 0,Y 510.553,Z 819.764,A -85,B 0,C 180,E1 -5398.225,E2 -5398.225} C_VEL
LIN {X 0,Y 510.799,Z 811.235,A -85,B 0,C 180,E1 -5398.916,E2 -5398.916} C_VEL
LIN {X 0,Y 511.031,Z 802.463,A -85,B 0,C 180,E1 -5399.507,E2 -5399.507} C_VEL
LIN {X 0,Y 511.316,Z 792.475,A -85,B 0,C 180,E1 -5400.049,E2 -5400.049} C_VEL
LIN {X 0,Y 511.532,Z 781.258,A -85,B 0,C 180,E1 -5400.516,E2 -5400.516} C_VEL
LIN {X 0,Y 511.62,Z 770.809,A -85,B 0,C 180,E1 -5400.836,E2 -5400.836} C_VEL
LIN {X 0,Y 511.782,Z 758.368,A -85,B 0,C 180,E1 -5401.082,E2 -5401.082} C_VEL
LIN {X 0,Y 512.016,Z 695.735,A -85,B 0,C 180,E1 -5401.985,E2 -5401.985} C_VEL
LIN {X 0,Y 510.213,Z 689.916,A -85,B 0,C 180,E1 -5402.146,E2 -5402.146} C_VEL
LIN {X 0,Y 510.075,Z 689.042,A -85,B 0,C 180,E1 -5402.295,E2 -5402.295} C_VEL
LIN {X 0,Y 509.978,Z 688.961,A -85,B 0,C 180,E1 -5405.536,E2 -5405.536} C_VEL
LIN {X 0,Y 509.91,Z 688.967,A -85,B 0,C 180,E1 -5408.72,E2 -5408.72} C_VEL
LIN {X 0,Y 509.912,Z 688.969,A -85,B 0,C 180,E1 -5411.931,E2 -5411.931} C_VEL
LIN {X 0,Y 509.902,Z 688.965,A -85,B 0,C 180,E1 -5415.242,E2 -5415.242} C_VEL
LIN {X 0,Y 509.867,Z 688.977,A -85,B 0,C 180,E1 -5418.483,E2 -5418.483} C_VEL
LIN {X 0,Y 509.857,Z 688.974,A -85,B 0,C 180,E1 -5421.001,E2 -5421.001} C_VEL
LIN {X 0,Y 509.864,Z 688.975,A -85,B 0,C 180,E1 -5424.426,E2 -5424.426} C_VEL
LIN {X 0,Y 509.866,Z 688.974,A -85,B 0,C 180,E1 -5427.057,E2 -5427.057} C_VEL
LIN {X 0,Y 509.864,Z 688.97,A -85,B 0,C 180,E1 -5429.751,E2 -5429.751} C_VEL
LIN {X 0,Y 509.873,Z 688.975,A -85,B 0,C 180,E1 -5432.772,E2 -5432.772} C_VEL
LIN {X 0,Y 509.832,Z 688.975,A -85,B 0,C 180,E1 -5435.578,E2 -5435.578} C_VEL
LIN {X 0,Y 509.856,Z 688.971,A -85,B 0,C 180,E1 -5438.338,E2 -5438.338} C_VEL
LIN {X 0,Y 509.862,Z 688.976,A -85,B 0,C 180,E1 -5441.425,E2 -5441.425} C_VEL
LIN {X 0,Y 509.845,Z 688.973,A -85,B 0,C 180,E1 -5444.669,E2 -5444.669} C_VEL
LIN {X 0,Y 509.862,Z 688.971,A -85,B 0,C 180,E1 -5448.103,E2 -5448.103} C_VEL
LIN {X 0,Y 509.84,Z 688.972,A -85,B 0,C 180,E1 -5450.646,E2 -5450.646} C_VEL
LIN {X 0,Y 509.815,Z 688.984,A -85,B 0,C 180,E1 -5453.645,E2 -5453.645} C_VEL
LIN {X 0,Y 509.847,Z 688.974,A -85,B 0,C 180,E1 -5456.537,E2 -5456.537} C_VEL
LIN {X 0,Y 509.851,Z 688.977,A -85,B 0,C 180,E1 -5459.334,E2 -5459.334} C_VEL
LIN {X 0,Y 509.905,Z 689.121,A -85,B 0,C 180,E1 -5460.733,E2 -5460.733} C_VEL
LIN {X 0,Y 513.171,Z 703.571,A -85,B 0,C 180,E1 -5462.753,E2 -5462.753} C_VEL
LIN {X 0,Y 512.684,Z 722.328,A -85,B 0,C 180,E1 -5465.068,E2 -5465.068} C_VEL
LIN {X 0,Y 511.914,Z 750.406,A -85,B 0,C 180,E1 -5468.474,E2 -5468.474} C_VEL
LIN {X 0,Y 511.289,Z 776.53,A -85,B 0,C 180,E1 -5471.569,E2 -5471.569} C_VEL
LIN {X 0,Y 510.783,Z 800.802,A -85,B 0,C 180,E1 -5474.398,E2 -5474.398} C_VEL
LIN {X 0,Y 512.221,Z 813.5,A -85,B 0,C 180,E1 -5474.633,E2 -5474.633} C_VEL
LIN {X 0,Y 511.746,Z 911.014,A -85,B 0,C 180,E1 -5476.017,E2 -5476.017} C_VEL
LIN {X 0,Y 511.515,Z 924.418,A -85,B 0,C 180,E1 -5476.365,E2 -5476.365} C_VEL
LIN {X 0,Y 511.172,Z 937.839,A -85,B 0,C 180,E1 -5476.887,E2 -5476.887} C_VEL
LIN {X 0,Y 510.896,Z 950.237,A -85,B 0,C 180,E1 -5477.555,E2 -5477.555} C_VEL
LIN {X 0,Y 510.594,Z 962.222,A -85,B 0,C 180,E1 -5478.386,E2 -5478.386} C_VEL
LIN {X 0,Y 510.248,Z 972.564,A -85,B 0,C 180,E1 -5479.283,E2 -5479.283} C_VEL
LIN {X 0,Y 509.968,Z 981.775,A -85,B 0,C 180,E1 -5480.28,E2 -5480.28} C_VEL
LIN {X 0,Y 509.669,Z 990.68,A -85,B 0,C 180,E1 -5481.474,E2 -5481.474} C_VEL
LIN {X 0,Y 509.439,Z 997.842,A -85,B 0,C 180,E1 -5482.667,E2 -5482.667} C_VEL
LIN {X 0,Y 509.371,Z 1004.361,A -85,B 0,C 180,E1 -5484.059,E2 -5484.059} C_VEL
LIN {X 0,Y 509.188,Z 1008.673,A -85,B 0,C 180,E1 -5485.249,E2 -5485.249} C_VEL
LIN {X 0,Y 509.253,Z 1010.955,A -85,B 0,C 180,E1 -5486.042,E2 -5486.042} C_VEL
LIN {X 0,Y 509.201,Z 1012.804,A -85,B 0,C 180,E1 -5486.834,E2 -5486.834} C_VEL
LIN {X 0,Y 509.161,Z 1014.191,A -85,B 0,C 180,E1 -5487.626,E2 -5487.626} C_VEL
LIN {X 0,Y 509.073,Z 1015.785,A -85,B 0,C 180,E1 -5489.208,E2 -5489.208} C_VEL
LIN {X 0,Y 509.065,Z 1016,A -85,B 0,C 180,E1 -5489.999,E2 -5489.999} C_VEL
LIN {X 0,Y 509.112,Z 1015.184,A -85,B 0,C 180,E1 -5491.581,E2 -5491.581} C_VEL
LIN {X 0,Y 509.16,Z 1014.197,A -85,B 0,C 180,E1 -5492.372,E2 -5492.372} C_VEL
LIN {X 0,Y 509.2,Z 1012.812,A -85,B 0,C 180,E1 -5493.164,E2 -5493.164} C_VEL
LIN {X 0,Y 509.233,Z 1009.898,A -85,B 0,C 180,E1 -5494.352,E2 -5494.352} C_VEL
LIN {X 0,Y 509.344,Z 1005.952,A -85,B 0,C 180,E1 -5495.541,E2 -5495.541} C_VEL
LIN {X 0,Y 509.401,Z 1000.333,A -85,B 0,C 180,E1 -5496.843,E2 -5496.843} C_VEL
LIN {X 0,Y 509.582,Z 993.243,A -85,B 0,C 180,E1 -5498.126,E2 -5498.126} C_VEL
LIN {X 0,Y 509.846,Z 985.001,A -85,B 0,C 180,E1 -5499.32,E2 -5499.32} C_VEL
LIN {X 0,Y 510.076,Z 976.52,A -85,B 0,C 180,E1 -5500.317,E2 -5500.317} C_VEL
LIN {X 0,Y 510.453,Z 965.923,A -85,B 0,C 180,E1 -5501.313,E2 -5501.313} C_VEL
LIN {X 0,Y 510.801,Z 954.422,A -85,B 0,C 180,E1 -5502.178,E2 -5502.178} C_VEL
LIN {X 0,Y 511.077,Z 943.868,A -85,B 0,C 180,E1 -5502.81,E2 -5502.81} C_VEL
LIN {X 0,Y 511.327,Z 932.063,A -85,B 0,C 180,E1 -5503.359,E2 -5503.359} C_VEL
LIN {X 0,Y 511.623,Z 918.517,A -85,B 0,C 180,E1 -5503.807,E2 -5503.807} C_VEL
LIN {X 0,Y 511.826,Z 905.166,A -85,B 0,C 180,E1 -5504.08,E2 -5504.08} C_VEL
LIN {X 0,Y 512.195,Z 811.959,A -85,B 0,C 180,E1 -5505.389,E2 -5505.389} C_VEL
LIN {X 0,Y 510.728,Z 800.447,A -85,B 0,C 180,E1 -5505.616,E2 -5505.616} C_VEL
LIN {X 0,Y 511.281,Z 774.758,A -85,B 0,C 180,E1 -5508.616,E2 -5508.616} C_VEL
LIN {X 0,Y 511.926,Z 749.93,A -85,B 0,C 180,E1 -5511.544,E2 -5511.544} C_VEL
LIN {X 0,Y 512.639,Z 721.933,A -85,B 0,C 180,E1 -5514.932,E2 -5514.932} C_VEL
LIN {X 0,Y 513.121,Z 703.695,A -85,B 0,C 180,E1 -5517.163,E2 -5517.163} C_VEL
LIN {X 0,Y 509.892,Z 689.109,A -85,B 0,C 180,E1 -5519.18,E2 -5519.18} C_VEL
LIN {X 0,Y 509.856,Z 688.979,A -85,B 0,C 180,E1 -5522.518,E2 -5522.518} C_VEL
LIN {X 0,Y 509.82,Z 688.977,A -85,B 0,C 180,E1 -5525.577,E2 -5525.577} C_VEL
LIN {X 0,Y 509.843,Z 688.978,A -85,B 0,C 180,E1 -5528.337,E2 -5528.337} C_VEL
LIN {X 0,Y 509.848,Z 688.972,A -85,B 0,C 180,E1 -5531.424,E2 -5531.424} C_VEL
LIN {X 0,Y 509.849,Z 688.979,A -85,B 0,C 180,E1 -5534.667,E2 -5534.667} C_VEL
LIN {X 0,Y 509.853,Z 688.972,A -85,B 0,C 180,E1 -5538.102,E2 -5538.102} C_VEL
LIN {X 0,Y 509.839,Z 688.973,A -85,B 0,C 180,E1 -5540.647,E2 -5540.647} C_VEL
LIN {X 0,Y 509.826,Z 688.972,A -85,B 0,C 180,E1 -5543.647,E2 -5543.647} C_VEL
LIN {X 0,Y 509.852,Z 688.971,A -85,B 0,C 180,E1 -5546.539,E2 -5546.539} C_VEL
LIN {X 0,Y 509.84,Z 688.98,A -85,B 0,C 180,E1 -5549.334,E2 -5549.334} C_VEL
LIN {X 0,Y 509.885,Z 688.966,A -85,B 0,C 180,E1 -5552.054,E2 -5552.054} C_VEL
LIN {X 0,Y 509.867,Z 688.968,A -85,B 0,C 180,E1 -5554.703,E2 -5554.703} C_VEL
LIN {X 0,Y 509.845,Z 688.979,A -85,B 0,C 180,E1 -5557.449,E2 -5557.449} C_VEL
LIN {X 0,Y 509.905,Z 688.97,A -85,B 0,C 180,E1 -5559.844,E2 -5559.844} C_VEL
LIN {X 0,Y 509.872,Z 688.967,A -85,B 0,C 180,E1 -5563.174,E2 -5563.174} C_VEL
LIN {X 0,Y 509.852,Z 688.977,A -85,B 0,C 180,E1 -5565.634,E2 -5565.634} C_VEL
LIN {X 0,Y 509.901,Z 688.964,A -85,B 0,C 180,E1 -5568.874,E2 -5568.874} C_VEL
LIN {X 0,Y 509.939,Z 688.965,A -85,B 0,C 180,E1 -5572.078,E2 -5572.078} C_VEL
LIN {X 0,Y 509.969,Z 688.959,A -85,B 0,C 180,E1 -5574.464,E2 -5574.464} C_VEL
LIN {X 0,Y 510.041,Z 688.947,A -85,B 0,C 180,E1 -5577.631,E2 -5577.631} C_VEL
LIN {X 0,Y 510.054,Z 688.948,A -85,B 0,C 180,E1 -5580.79,E2 -5580.79} C_VEL
LIN {X 0,Y 509.945,Z 688.959,A -85,B 0,C 180,E1 -5583.16,E2 -5583.16} C_VEL
LIN {X 0,Y 509.941,Z 688.964,A -85,B 0,C 180,E1 -5586.33,E2 -5586.33} C_VEL
LIN {X 0,Y 509.905,Z 688.97,A -85,B 0,C 180,E1 -5588.721,E2 -5588.721} C_VEL
LIN {X 0,Y 509.893,Z 688.964,A -85,B 0,C 180,E1 -5591.932,E2 -5591.932} C_VEL
LIN {X 0,Y 509.882,Z 688.969,A -85,B 0,C 180,E1 -5595.242,E2 -5595.242} C_VEL
LIN {X 0,Y 509.85,Z 688.973,A -85,B 0,C 180,E1 -5598.484,E2 -5598.484} C_VEL
LIN {X 0,Y 509.839,Z 688.98,A -85,B 0,C 180,E1 -5601.002,E2 -5601.002} C_VEL
LIN {X 0,Y 509.809,Z 688.976,A -85,B 0,C 180,E1 -5603.565,E2 -5603.565} C_VEL
LIN {X 0,Y 509.876,Z 688.969,A -85,B 0,C 180,E1 -5606.374,E2 -5606.374} C_VEL
LIN {X 0,Y 509.862,Z 688.967,A -85,B 0,C 180,E1 -5608.845,E2 -5608.845} C_VEL
LIN {X 0,Y 509.812,Z 688.981,A -85,B 0,C 180,E1 -5611.591,E2 -5611.591} C_VEL
LIN {X 0,Y 509.843,Z 688.973,A -85,B 0,C 180,E1 -5614.414,E2 -5614.414} C_VEL
LIN {X 0,Y 509.81,Z 688.98,A -85,B 0,C 180,E1 -5617.342,E2 -5617.342} C_VEL
LIN {X 0,Y 509.831,Z 688.975,A -85,B 0,C 180,E1 -5620.383,E2 -5620.383} C_VEL
LIN {X 0,Y 509.816,Z 688.976,A -85,B 0,C 180,E1 -5623.063,E2 -5623.063} C_VEL
LIN {X 0,Y 509.816,Z 688.983,A -85,B 0,C 180,E1 -5625.795,E2 -5625.795} C_VEL
LIN {X 0,Y 509.847,Z 688.973,A -85,B 0,C 180,E1 -5628.576,E2 -5628.576} C_VEL
LIN {X 0,Y 509.899,Z 689.148,A -85,B 0,C 180,E1 -5629.732,E2 -5629.732} C_VEL
LIN {X 0,Y 510.074,Z 690.046,A -85,B 0,C 180,E1 -5629.856,E2 -5629.856} C_VEL
LIN {X 0,Y 512.332,Z 696.693,A -85,B 0,C 180,E1 -5630.04,E2 -5630.04} C_VEL
LIN {X 0,Y 512.205,Z 717.211,A -85,B 0,C 180,E1 -5630.331,E2 -5630.331} C_VEL
LIN {X 0,Y 511.417,Z 723.054,A -85,B 0,C 180,E1 -5630.39,E2 -5630.39} C_VEL
LIN {X 0,Y 505.833,Z 742.061,A -85,B 0,C 180,E1 -5630.489,E2 -5630.489} C_VEL
LIN {X 0,Y 505.178,Z 747.9,A -85,B 0,C 180,E1 -5630.553,E2 -5630.553} C_VEL
LIN {X 0,Y 505.094,Z 771.827,A -85,B 0,C 180,E1 -5630.932,E2 -5630.932} C_VEL
LIN {X 0,Y 505.015,Z 784.803,A -85,B 0,C 180,E1 -5631.304,E2 -5631.304} C_VEL
LIN {X 0,Y 504.859,Z 796.407,A -85,B 0,C 180,E1 -5631.788,E2 -5631.788} C_VEL
LIN {X 0,Y 504.643,Z 807.999,A -85,B 0,C 180,E1 -5632.437,E2 -5632.437} C_VEL
LIN {X 0,Y 504.273,Z 819.929,A -85,B 0,C 180,E1 -5633.297,E2 -5633.297} C_VEL
LIN {X 0,Y 503.958,Z 830.537,A -85,B 0,C 180,E1 -5634.271,E2 -5634.271} C_VEL
LIN {X 0,Y 503.595,Z 839.681,A -85,B 0,C 180,E1 -5635.315,E2 -5635.315} C_VEL
LIN {X 0,Y 503.267,Z 848.251,A -85,B 0,C 180,E1 -5636.525,E2 -5636.525} C_VEL
LIN {X 0,Y 503.074,Z 854.915,A -85,B 0,C 180,E1 -5637.701,E2 -5637.701} C_VEL
LIN {X 0,Y 502.847,Z 860.215,A -85,B 0,C 180,E1 -5638.862,E2 -5638.862} C_VEL
LIN {X 0,Y 502.693,Z 864.623,A -85,B 0,C 180,E1 -5640.09,E2 -5640.09} C_VEL
LIN {X 0,Y 502.601,Z 867.573,A -85,B 0,C 180,E1 -5641.158,E2 -5641.158} C_VEL
LIN {X 0,Y 502.494,Z 870.224,A -85,B 0,C 180,E1 -5642.515,E2 -5642.515} C_VEL
LIN {X 0,Y 502.462,Z 871.425,A -85,B 0,C 180,E1 -5643.532,E2 -5643.532} C_VEL
LIN {X 0,Y 502.441,Z 871.948,A -85,B 0,C 180,E1 -5644.304,E2 -5644.304} C_VEL
LIN {X 0,Y 502.416,Z 872.045,A -85,B 0,C 180,E1 -5645.402,E2 -5645.402} C_VEL
LIN {X 0,Y 502.447,Z 870.998,A -85,B 0,C 180,E1 -5646.944,E2 -5646.944} C_VEL
LIN {X 0,Y 502.484,Z 869.738,A -85,B 0,C 180,E1 -5647.814,E2 -5647.814} C_VEL
LIN {X 0,Y 502.641,Z 866.975,A -85,B 0,C 180,E1 -5649.114,E2 -5649.114} C_VEL
LIN {X 0,Y 502.736,Z 863.136,A -85,B 0,C 180,E1 -5650.398,E2 -5650.398} C_VEL
LIN {X 0,Y 502.937,Z 857.325,A -85,B 0,C 180,E1 -5651.848,E2 -5651.848} C_VEL
LIN {X 0,Y 503.158,Z 850.478,A -85,B 0,C 180,E1 -5653.154,E2 -5653.154} C_VEL
LIN {X 0,Y 503.458,Z 842.178,A -85,B 0,C 180,E1 -5654.41,E2 -5654.41} C_VEL
LIN {X 0,Y 503.728,Z 833.643,A -85,B 0,C 180,E1 -5655.457,E2 -5655.457} C_VEL
LIN {X 0,Y 504.103,Z 823.039,A -85,B 0,C 180,E1 -5656.497,E2 -5656.497} C_VEL
LIN {X 0,Y 504.448,Z 811.819,A -85,B 0,C 180,E1 -5657.375,E2 -5657.375} C_VEL
LIN {X 0,Y 504.696,Z 800.954,A -85,B 0,C 180,E1 -5658.047,E2 -5658.047} C_VEL
LIN {X 0,Y 504.918,Z 788.911,A -85,B 0,C 180,E1 -5658.612,E2 -5658.612} C_VEL
LIN {X 0,Y 505.047,Z 775.905,A -85,B 0,C 180,E1 -5659.047,E2 -5659.047} C_VEL
LIN {X 0,Y 505.14,Z 763.541,A -85,B 0,C 180,E1 -5659.302,E2 -5659.302} C_VEL
LIN {X 0,Y 505.37,Z 697.585,A -85,B 0,C 180,E1 -5660.253,E2 -5660.253} C_VEL
LIN {X 0,Y 503.023,Z 690.786,A -85,B 0,C 180,E1 -5660.451,E2 -5660.451} C_VEL
LIN {X 0,Y 502.843,Z 689.945,A -85,B 0,C 180,E1 -5660.6,E2 -5660.6} C_VEL
LIN {X 0,Y 502.875,Z 689.841,A -85,B 0,C 180,E1 -5663.582,E2 -5663.582} C_VEL
LIN {X 0,Y 502.833,Z 689.849,A -85,B 0,C 180,E1 -5666.796,E2 -5666.796} C_VEL
LIN {X 0,Y 502.896,Z 689.845,A -85,B 0,C 180,E1 -5668.4,E2 -5668.4} C_VEL
LIN {X 0,Y 503.006,Z 689.83,A -85,B 0,C 180,E1 -5670.001,E2 -5670.001} C_VEL
LIN {X 0,Y 503.01,Z 689.831,A -85,B 0,C 180,E1 -5672.403,E2 -5672.403} C_VEL
LIN {X 0,Y 502.897,Z 689.839,A -85,B 0,C 180,E1 -5675.615,E2 -5675.615} C_VEL
LIN {X 0,Y 502.851,Z 689.844,A -85,B 0,C 180,E1 -5678.035,E2 -5678.035} C_VEL
LIN {X 0,Y 502.837,Z 689.844,A -85,B 0,C 180,E1 -5681.285,E2 -5681.285} C_VEL
LIN {X 0,Y 502.832,Z 689.85,A -85,B 0,C 180,E1 -5684.572,E2 -5684.572} C_VEL
LIN {X 0,Y 502.791,Z 689.85,A -85,B 0,C 180,E1 -5687.911,E2 -5687.911} C_VEL
LIN {X 0,Y 502.809,Z 689.847,A -85,B 0,C 180,E1 -5690.528,E2 -5690.528} C_VEL
LIN {X 0,Y 502.79,Z 689.858,A -85,B 0,C 180,E1 -5693.042,E2 -5693.042} C_VEL
LIN {X 0,Y 502.762,Z 689.849,A -85,B 0,C 180,E1 -5695.681,E2 -5695.681} C_VEL
LIN {X 0,Y 502.765,Z 689.85,A -85,B 0,C 180,E1 -5698.378,E2 -5698.378} C_VEL
LIN {X 0,Y 502.771,Z 689.856,A -85,B 0,C 180,E1 -5701.494,E2 -5701.494} C_VEL
LIN {X 0,Y 502.777,Z 689.843,A -85,B 0,C 180,E1 -5704.439,E2 -5704.439} C_VEL
LIN {X 0,Y 502.724,Z 689.858,A -85,B 0,C 180,E1 -5707.169,E2 -5707.169} C_VEL
LIN {X 0,Y 502.735,Z 689.859,A -85,B 0,C 180,E1 -5710.021,E2 -5710.021} C_VEL
LIN {X 0,Y 502.74,Z 689.861,A -85,B 0,C 180,E1 -5713.236,E2 -5713.236} C_VEL
LIN {X 0,Y 502.774,Z 689.861,A -85,B 0,C 180,E1 -5715.659,E2 -5715.659} C_VEL
LIN {X 0,Y 502.756,Z 689.855,A -85,B 0,C 180,E1 -5719.015,E2 -5719.015} C_VEL
LIN {X 0,Y 502.744,Z 689.863,A -85,B 0,C 180,E1 -5722.041,E2 -5722.041} C_VEL
LIN {X 0,Y 502.756,Z 689.855,A -85,B 0,C 180,E1 -5725.03,E2 -5725.03} C_VEL
LIN {X 0,Y 502.762,Z 689.862,A -85,B 0,C 180,E1 -5727.914,E2 -5727.914} C_VEL
LIN {X 0,Y 502.763,Z 689.859,A -85,B 0,C 180,E1 -5731.166,E2 -5731.166} C_VEL
LIN {X 0,Y 502.807,Z 690.123,A -85,B 0,C 180,E1 -5731.645,E2 -5731.645} C_VEL
LIN {X 0,Y 503.09,Z 691.296,A -85,B 0,C 180,E1 -5731.76,E2 -5731.76} C_VEL
LIN {X 0,Y 505.179,Z 697.379,A -85,B 0,C 180,E1 -5731.922,E2 -5731.922} C_VEL
LIN {X 0,Y 504.821,Z 765.458,A -85,B 0,C 180,E1 -5732.938,E2 -5732.938} C_VEL
LIN {X 0,Y 504.664,Z 777.227,A -85,B 0,C 180,E1 -5733.244,E2 -5733.244} C_VEL
LIN {X 0,Y 504.476,Z 787.775,A -85,B 0,C 180,E1 -5733.637,E2 -5733.637} C_VEL
LIN {X 0,Y 504.291,Z 796.835,A -85,B 0,C 180,E1 -5734.071,E2 -5734.071} C_VEL
LIN {X 0,Y 504.01,Z 806.967,A -85,B 0,C 180,E1 -5734.683,E2 -5734.683} C_VEL
LIN {X 0,Y 503.755,Z 816.179,A -85,B 0,C 180,E1 -5735.367,E2 -5735.367} C_VEL
LIN {X 0,Y 503.442,Z 824.604,A -85,B 0,C 180,E1 -5736.119,E2 -5736.119} C_VEL
LIN {X 0,Y 503.247,Z 832.647,A -85,B 0,C 180,E1 -5736.981,E2 -5736.981} C_VEL
LIN {X 0,Y 503.024,Z 839.443,A -85,B 0,C 180,E1 -5737.837,E2 -5737.837} C_VEL
LIN {X 0,Y 502.709,Z 846.565,A -85,B 0,C 180,E1 -5738.922,E2 -5738.922} C_VEL
LIN {X 0,Y 502.587,Z 852.219,A -85,B 0,C 180,E1 -5739.964,E2 -5739.964} C_VEL
LIN {X 0,Y 502.429,Z 857.71,A -85,B 0,C 180,E1 -5741.232,E2 -5741.232} C_VEL
LIN {X 0,Y 502.365,Z 860.755,A -85,B 0,C 180,E1 -5742.075,E2 -5742.075} C_VEL
LIN {X 0,Y 502.201,Z 865.032,A -85,B 0,C 180,E1 -5743.746,E2 -5743.746} C_VEL
LIN {X 0,Y 502.151,Z 867.054,A -85,B 0,C 180,E1 -5744.955,E2 -5744.955} C_VEL
LIN {X 0,Y 502.171,Z 868.264,A -85,B 0,C 180,E1 -5746.236,E2 -5746.236} C_VEL
LIN {X 0,Y 502.167,Z 868.511,A -85,B 0,C 180,E1 -5747.06,E2 -5747.06} C_VEL
LIN {X 0,Y 502.233,Z 867.97,A -85,B 0,C 180,E1 -5748.395,E2 -5748.395} C_VEL
LIN {X 0,Y 502.254,Z 866.704,A -85,B 0,C 180,E1 -5749.519,E2 -5749.519} C_VEL
LIN {X 0,Y 502.262,Z 865.241,A -85,B 0,C 180,E1 -5750.333,E2 -5750.333} C_VEL
LIN {X 0,Y 502.38,Z 861.146,A -85,B 0,C 180,E1 -5751.958,E2 -5751.958} C_VEL
LIN {X 0,Y 502.547,Z 856.755,A -85,B 0,C 180,E1 -5753.184,E2 -5753.184} C_VEL
LIN {X 0,Y 502.678,Z 850.148,A -85,B 0,C 180,E1 -5754.585,E2 -5754.585} C_VEL
LIN {X 0,Y 502.859,Z 844.291,A -85,B 0,C 180,E1 -5755.591,E2 -5755.591} C_VEL
LIN {X 0,Y 503.086,Z 837.237,A -85,B 0,C 180,E1 -5756.596,E2 -5756.596} C_VEL
LIN {X 0,Y 503.348,Z 830.58,A -85,B 0,C 180,E1 -5757.399,E2 -5757.399} C_VEL
LIN {X 0,Y 503.628,Z 821.571,A -85,B 0,C 180,E1 -5758.301,E2 -5758.301} C_VEL
LIN {X 0,Y 503.922,Z 811.789,A -85,B 0,C 180,E1 -5759.101,E2 -5759.101} C_VEL
LIN {X 0,Y 504.158,Z 802.889,A -85,B 0,C 180,E1 -5759.7,E2 -5759.7} C_VEL
LIN {X 0,Y 504.454,Z 792.709,A -85,B 0,C 180,E1 -5760.249,E2 -5760.249} C_VEL
LIN {X 0,Y 504.647,Z 782.661,A -85,B 0,C 180,E1 -5760.673,E2 -5760.673} C_VEL
LIN {X 0,Y 504.723,Z 772.368,A -85,B 0,C 180,E1 -5760.997,E2 -5760.997} C_VEL
LIN {X 0,Y 504.895,Z 760.188,A -85,B 0,C 180,E1 -5761.246,E2 -5761.246} C_VEL
LIN {X 0,Y 505.117,Z 696.899,A -85,B 0,C 180,E1 -5762.18,E2 -5762.18} C_VEL
LIN {X 0,Y 503.203,Z 690.807,A -85,B 0,C 180,E1 -5762.351,E2 -5762.351} C_VEL
LIN {X 0,Y 502.999,Z 689.928,A -85,B 0,C 180,E1 -5762.502,E2 -5762.502} C_VEL
LIN {X 0,Y 502.931,Z 689.839,A -85,B 0,C 180,E1 -5765.613,E2 -5765.613} C_VEL
LIN {X 0,Y 502.87,Z 689.844,A -85,B 0,C 180,E1 -5768.843,E2 -5768.843} C_VEL
LIN {X 0,Y 502.852,Z 689.849,A -85,B 0,C 180,E1 -5772.101,E2 -5772.101} C_VEL
LIN {X 0,Y 502.856,Z 689.843,A -85,B 0,C 180,E1 -5775.399,E2 -5775.399} C_VEL
LIN {X 0,Y 502.833,Z 689.851,A -85,B 0,C 180,E1 -5778.752,E2 -5778.752} C_VEL
LIN {X 0,Y 502.79,Z 689.852,A -85,B 0,C 180,E1 -5781.311,E2 -5781.311} C_VEL
LIN {X 0,Y 502.788,Z 689.851,A -85,B 0,C 180,E1 -5783.914,E2 -5783.914} C_VEL
LIN {X 0,Y 502.842,Z 689.852,A -85,B 0,C 180,E1 -5786.567,E2 -5786.567} C_VEL
LIN {X 0,Y 502.822,Z 689.847,A -85,B 0,C 180,E1 -5789.935,E2 -5789.935} C_VEL
LIN {X 0,Y 502.836,Z 689.853,A -85,B 0,C 180,E1 -5793.031,E2 -5793.031} C_VEL
LIN {X 0,Y 502.78,Z 689.852,A -85,B 0,C 180,E1 -5795.951,E2 -5795.951} C_VEL
LIN {X 0,Y 502.807,Z 689.855,A -85,B 0,C 180,E1 -5798.976,E2 -5798.976} C_VEL
LIN {X 0,Y 502.801,Z 689.85,A -85,B 0,C 180,E1 -5802.139,E2 -5802.139} C_VEL
LIN {X 0,Y 502.792,Z 689.858,A -85,B 0,C 180,E1 -5805.469,E2 -5805.469} C_VEL
LIN {X 0,Y 502.826,Z 689.849,A -85,B 0,C 180,E1 -5808.933,E2 -5808.933} C_VEL
LIN {X 0,Y 502.796,Z 689.852,A -85,B 0,C 180,E1 -5812.045,E2 -5812.045} C_VEL
LIN {X 0,Y 502.8,Z 689.852,A -85,B 0,C 180,E1 -5815.033,E2 -5815.033} C_VEL
LIN {X 0,Y 502.788,Z 689.858,A -85,B 0,C 180,E1 -5817.915,E2 -5817.915} C_VEL
LIN {X 0,Y 502.89,Z 690.004,A -85,B 0,C 180,E1 -5820.511,E2 -5820.511} C_VEL
LIN {X 0,Y 506.359,Z 705.789,A -85,B 0,C 180,E1 -5822.739,E2 -5822.739} C_VEL
LIN {X 0,Y 505.621,Z 728.473,A -85,B 0,C 180,E1 -5825.573,E2 -5825.573} C_VEL
LIN {X 0,Y 504.846,Z 754.552,A -85,B 0,C 180,E1 -5828.779,E2 -5828.779} C_VEL
LIN {X 0,Y 504.142,Z 782.6,A -85,B 0,C 180,E1 -5832.139,E2 -5832.139} C_VEL
LIN {X 0,Y 503.733,Z 799.785,A -85,B 0,C 180,E1 -5834.172,E2 -5834.172} C_VEL
LIN {X 0,Y 505.344,Z 813.653,A -85,B 0,C 180,E1 -5834.435,E2 -5834.435} C_VEL
LIN {X 0,Y 504.857,Z 909.961,A -85,B 0,C 180,E1 -5835.822,E2 -5835.822} C_VEL
LIN {X 0,Y 504.551,Z 923.378,A -85,B 0,C 180,E1 -5836.173,E2 -5836.173} C_VEL
LIN {X 0,Y 504.235,Z 936.815,A -85,B 0,C 180,E1 -5836.703,E2 -5836.703} C_VEL
LIN {X 0,Y 503.929,Z 948.63,A -85,B 0,C 180,E1 -5837.342,E2 -5837.342} C_VEL
LIN {X 0,Y 503.613,Z 959.892,A -85,B 0,C 180,E1 -5838.12,E2 -5838.12} C_VEL
LIN {X 0,Y 503.223,Z 970.497,A -85,B 0,C 180,E1 -5839.029,E2 -5839.029} C_VEL
LIN {X 0,Y 502.961,Z 979.196,A -85,B 0,C 180,E1 -5839.94,E2 -5839.94} C_VEL
LIN {X 0,Y 502.696,Z 987.233,A -85,B 0,C 180,E1 -5840.95,E2 -5840.95} C_VEL
LIN {X 0,Y 502.445,Z 995.1,A -85,B 0,C 180,E1 -5842.16,E2 -5842.16} C_VEL
LIN {X 0,Y 502.276,Z 1002.365,A -85,B 0,C 180,E1 -5843.572,E2 -5843.572} C_VEL
LIN {X 0,Y 502.186,Z 1007.203,A -85,B 0,C 180,E1 -5844.78,E2 -5844.78} C_VEL
LIN {X 0,Y 502.15,Z 1010.875,A -85,B 0,C 180,E1 -5845.986,E2 -5845.986} C_VEL
LIN {X 0,Y 502.121,Z 1012.755,A -85,B 0,C 180,E1 -5846.789,E2 -5846.789} C_VEL
LIN {X 0,Y 502.065,Z 1014.159,A -85,B 0,C 180,E1 -5847.592,E2 -5847.592} C_VEL
LIN {X 0,Y 502.035,Z 1015.158,A -85,B 0,C 180,E1 -5848.394,E2 -5848.394} C_VEL
LIN {X 0,Y 501.98,Z 1015.984,A -85,B 0,C 180,E1 -5849.999,E2 -5849.999} C_VEL
LIN {X 0,Y 502.035,Z 1015.163,A -85,B 0,C 180,E1 -5851.603,E2 -5851.603} C_VEL
LIN {X 0,Y 502.065,Z 1014.165,A -85,B 0,C 180,E1 -5852.406,E2 -5852.406} C_VEL
LIN {X 0,Y 502.12,Z 1012.764,A -85,B 0,C 180,E1 -5853.208,E2 -5853.208} C_VEL
LIN {X 0,Y 502.125,Z 1009.794,A -85,B 0,C 180,E1 -5854.414,E2 -5854.414} C_VEL
LIN {X 0,Y 502.259,Z 1005.754,A -85,B 0,C 180,E1 -5855.62,E2 -5855.62} C_VEL
LIN {X 0,Y 502.332,Z 999.585,A -85,B 0,C 180,E1 -5857.01,E2 -5857.01} C_VEL
LIN {X 0,Y 502.512,Z 992.648,A -85,B 0,C 180,E1 -5858.241,E2 -5858.241} C_VEL
LIN {X 0,Y 502.794,Z 984.189,A -85,B 0,C 180,E1 -5859.452,E2 -5859.452} C_VEL
LIN {X 0,Y 503.062,Z 975.524,A -85,B 0,C 180,E1 -5860.463,E2 -5860.463} C_VEL
LIN {X 0,Y 503.429,Z 964.85,A -85,B 0,C 180,E1 -5861.473,E2 -5861.473} C_VEL
LIN {X 0,Y 503.763,Z 953.336,A -85,B 0,C 180,E1 -5862.351,E2 -5862.351} C_VEL
LIN {X 0,Y 504.079,Z 942.777,A -85,B 0,C 180,E1 -5862.991,E2 -5862.991} C_VEL
LIN {X 0,Y 504.388,Z 930.963,A -85,B 0,C 180,E1 -5863.547,E2 -5863.547} C_VEL
LIN {X 0,Y 504.691,Z 917.398,A -85,B 0,C 180,E1 -5864,E2 -5864} C_VEL
LIN {X 0,Y 504.9,Z 903.999,A -85,B 0,C 180,E1 -5864.277,E2 -5864.277} C_VEL
LIN {X 0,Y 505.268,Z 812.313,A -85,B 0,C 180,E1 -5865.584,E2 -5865.584} C_VEL
LIN {X 0,Y 503.704,Z 799.393,A -85,B 0,C 180,E1 -5865.838,E2 -5865.838} C_VEL
LIN {X 0,Y 504.28,Z 773.554,A -85,B 0,C 180,E1 -5868.905,E2 -5868.905} C_VEL
LIN {X 0,Y 504.946,Z 748.946,A -85,B 0,C 180,E1 -5871.857,E2 -5871.857} C_VEL
LIN {X 0,Y 505.736,Z 721.827,A -85,B 0,C 180,E1 -5875.185,E2 -5875.185} C_VEL
LIN {X 0,Y 506.178,Z 704.866,A -85,B 0,C 180,E1 -5877.301,E2 -5877.301} C_VEL
LIN {X 0,Y 502.881,Z 690.018,A -85,B 0,C 180,E1 -5879.385,E2 -5879.385} C_VEL
LIN {X 0,Y 502.778,Z 689.855,A -85,B 0,C 180,E1 -5882.083,E2 -5882.083} C_VEL
LIN {X 0,Y 502.793,Z 689.854,A -85,B 0,C 180,E1 -5884.965,E2 -5884.965} C_VEL
LIN {X 0,Y 502.786,Z 689.854,A -85,B 0,C 180,E1 -5887.953,E2 -5887.953} C_VEL
LIN {X 0,Y 502.812,Z 689.852,A -85,B 0,C 180,E1 -5891.065,E2 -5891.065} C_VEL
LIN {X 0,Y 502.793,Z 689.856,A -85,B 0,C 180,E1 -5894.531,E2 -5894.531} C_VEL
LIN {X 0,Y 502.822,Z 689.847,A -85,B 0,C 180,E1 -5897.863,E2 -5897.863} C_VEL
LIN {X 0,Y 502.794,Z 689.855,A -85,B 0,C 180,E1 -5901.023,E2 -5901.023} C_VEL
LIN {X 0,Y 502.776,Z 689.848,A -85,B 0,C 180,E1 -5904.166,E2 -5904.166} C_VEL
LIN {X 0,Y 502.822,Z 689.852,A -85,B 0,C 180,E1 -5906.992,E2 -5906.992} C_VEL
LIN {X 0,Y 502.82,Z 689.847,A -85,B 0,C 180,E1 -5910.061,E2 -5910.061} C_VEL
LIN {X 0,Y 502.825,Z 689.845,A -85,B 0,C 180,E1 -5912.533,E2 -5912.533} C_VEL
LIN {X 0,Y 502.818,Z 689.852,A -85,B 0,C 180,E1 -5915.298,E2 -5915.298} C_VEL
LIN {X 0,Y 502.782,Z 689.854,A -85,B 0,C 180,E1 -5917.827,E2 -5917.827} C_VEL
LIN {X 0,Y 502.813,Z 689.848,A -85,B 0,C 180,E1 -5920.4,E2 -5920.4} C_VEL
LIN {X 0,Y 502.821,Z 689.843,A -85,B 0,C 180,E1 -5922.931,E2 -5922.931} C_VEL
LIN {X 0,Y 502.833,Z 689.848,A -85,B 0,C 180,E1 -5925.429,E2 -5925.429} C_VEL
LIN {X 0,Y 502.865,Z 689.841,A -85,B 0,C 180,E1 -5928.717,E2 -5928.717} C_VEL
LIN {X 0,Y 502.889,Z 689.841,A -85,B 0,C 180,E1 -5931.967,E2 -5931.967} C_VEL
LIN {X 0,Y 502.922,Z 689.837,A -85,B 0,C 180,E1 -5934.386,E2 -5934.386} C_VEL
LIN {X 0,Y 503.011,Z 689.823,A -85,B 0,C 180,E1 -5937.598,E2 -5937.598} C_VEL
LIN {X 0,Y 503.013,Z 689.825,A -85,B 0,C 180,E1 -5940,E2 -5940} C_VEL
LIN {X 0,Y 503.012,Z 689.831,A -85,B 0,C 180,E1 -5942.402,E2 -5942.402} C_VEL
LIN {X 0,Y 502.923,Z 689.833,A -85,B 0,C 180,E1 -5945.614,E2 -5945.614} C_VEL
LIN {X 0,Y 502.89,Z 689.838,A -85,B 0,C 180,E1 -5948.034,E2 -5948.034} C_VEL
LIN {X 0,Y 502.869,Z 689.841,A -85,B 0,C 180,E1 -5951.284,E2 -5951.284} C_VEL
LIN {X 0,Y 502.832,Z 689.85,A -85,B 0,C 180,E1 -5954.571,E2 -5954.571} C_VEL
LIN {X 0,Y 502.811,Z 689.848,A -85,B 0,C 180,E1 -5957.909,E2 -5957.909} C_VEL
LIN {X 0,Y 502.818,Z 689.848,A -85,B 0,C 180,E1 -5960.537,E2 -5960.537} C_VEL
LIN {X 0,Y 502.776,Z 689.854,A -85,B 0,C 180,E1 -5963.042,E2 -5963.042} C_VEL
LIN {X 0,Y 502.834,Z 689.846,A -85,B 0,C 180,E1 -5966.558,E2 -5966.558} C_VEL
LIN {X 0,Y 502.812,Z 689.85,A -85,B 0,C 180,E1 -5969.289,E2 -5969.289} C_VEL
LIN {X 0,Y 502.775,Z 689.851,A -85,B 0,C 180,E1 -5972.086,E2 -5972.086} C_VEL
LIN {X 0,Y 502.798,Z 689.851,A -85,B 0,C 180,E1 -5974.966,E2 -5974.966} C_VEL
LIN {X 0,Y 502.785,Z 689.855,A -85,B 0,C 180,E1 -5977.955,E2 -5977.955} C_VEL
LIN {X 0,Y 502.813,Z 689.849,A -85,B 0,C 180,E1 -5981.067,E2 -5981.067} C_VEL
LIN {X 0,Y 502.779,Z 689.856,A -85,B 0,C 180,E1 -5984.531,E2 -5984.531} C_VEL
LIN {X 0,Y 502.788,Z 689.858,A -85,B 0,C 180,E1 -5987.862,E2 -5987.862} C_VEL
LIN {X 0,Y 502.83,Z 690.053,A -85,B 0,C 180,E1 -5989.514,E2 -5989.514} C_VEL
LIN {X 0,Y 503.117,Z 691.217,A -85,B 0,C 180,E1 -5989.649,E2 -5989.649} C_VEL
LIN {X 0,Y 505.416,Z 697.594,A -85,B 0,C 180,E1 -5989.827,E2 -5989.827} C_VEL
LIN {X 0,Y 505.178,Z 747.9,A -85,B 0,C 180,E1 -5990.553,E2 -5990.553} C_VEL
LIN {X 0,Y 504.506,Z 753.752,A -85,B 0,C 180,E1 -5990.614,E2 -5990.614} C_VEL
LIN {X 0,Y 498.909,Z 772.725,A -85,B 0,C 180,E1 -5990.752,E2 -5990.752} C_VEL
LIN {X 0,Y 498.24,Z 778.469,A -85,B 0,C 180,E1 -5990.878,E2 -5990.878} C_VEL
LIN {X 0,Y 498.081,Z 791.315,A -85,B 0,C 180,E1 -5991.325,E2 -5991.325} C_VEL
LIN {X 0,Y 497.88,Z 802.95,A -85,B 0,C 180,E1 -5991.891,E2 -5991.891} C_VEL
LIN {X 0,Y 497.612,Z 814.137,A -85,B 0,C 180,E1 -5992.607,E2 -5992.607} C_VEL
LIN {X 0,Y 497.267,Z 824.774,A -85,B 0,C 180,E1 -5993.463,E2 -5993.463} C_VEL
LIN {X 0,Y 496.95,Z 834.534,A -85,B 0,C 180,E1 -5994.439,E2 -5994.439} C_VEL
LIN {X 0,Y 496.555,Z 843.306,A -85,B 0,C 180,E1 -5995.52,E2 -5995.52} C_VEL
LIN {X 0,Y 496.274,Z 850.869,A -85,B 0,C 180,E1 -5996.672,E2 -5996.672} C_VEL
LIN {X 0,Y 496.037,Z 857.298,A -85,B 0,C 180,E1 -5997.881,E2 -5997.881} C_VEL
LIN {X 0,Y 495.774,Z 863.304,A -85,B 0,C 180,E1 -5999.316,E2 -5999.316} C_VEL
LIN {X 0,Y 495.662,Z 867.607,A -85,B 0,C 180,E1 -6000.715,E2 -6000.715} C_VEL
LIN {X 0,Y 495.498,Z 870.594,A -85,B 0,C 180,E1 -6002.093,E2 -6002.093} C_VEL
LIN {X 0,Y 495.461,Z 872.273,A -85,B 0,C 180,E1 -6003.335,E2 -6003.335} C_VEL
LIN {X 0,Y 495.395,Z 873.088,A -85,B 0,C 180,E1 -6004.813,E2 -6004.813} C_VEL
LIN {X 0,Y 495.386,Z 872.984,A -85,B 0,C 180,E1 -6005.707,E2 -6005.707} C_VEL
LIN {X 0,Y 495.446,Z 871.668,A -85,B 0,C 180,E1 -6007.227,E2 -6007.227} C_VEL
LIN {X 0,Y 495.567,Z 868.872,A -85,B 0,C 180,E1 -6008.801,E2 -6008.801} C_VEL
LIN {X 0,Y 495.695,Z 865.348,A -85,B 0,C 180,E1 -6010.108,E2 -6010.108} C_VEL
LIN {X 0,Y 495.917,Z 860.452,A -85,B 0,C 180,E1 -6011.45,E2 -6011.45} C_VEL
LIN {X 0,Y 496.092,Z 854.622,A -85,B 0,C 180,E1 -6012.694,E2 -6012.694} C_VEL
LIN {X 0,Y 496.378,Z 846.81,A -85,B 0,C 180,E1 -6014.016,E2 -6014.016} C_VEL
LIN {X 0,Y 496.676,Z 839.371,A -85,B 0,C 180,E1 -6015.036,E2 -6015.036} C_VEL
LIN {X 0,Y 497.023,Z 829.985,A -85,B 0,C 180,E1 -6016.092,E2 -6016.092} C_VEL
LIN {X 0,Y 497.353,Z 819.462,A -85,B 0,C 180,E1 -6017.042,E2 -6017.042} C_VEL
LIN {X 0,Y 497.685,Z 807.854,A -85,B 0,C 180,E1 -6017.876,E2 -6017.876} C_VEL
LIN {X 0,Y 497.942,Z 795.509,A -85,B 0,C 180,E1 -6018.553,E2 -6018.553} C_VEL
LIN {X 0,Y 498.149,Z 782.463,A -85,B 0,C 180,E1 -6019.073,E2 -6019.073} C_VEL
LIN {X 0,Y 498.269,Z 769.694,A -85,B 0,C 180,E1 -6019.41,E2 -6019.41} C_VEL
LIN {X 0,Y 498.507,Z 698.844,A -85,B 0,C 180,E1 -6020.46,E2 -6020.46} C_VEL
LIN {X 0,Y 496.005,Z 691.809,A -85,B 0,C 180,E1 -6020.665,E2 -6020.665} C_VEL
LIN {X 0,Y 495.811,Z 690.833,A -85,B 0,C 180,E1 -6020.82,E2 -6020.82} C_VEL
LIN {X 0,Y 495.826,Z 690.718,A -85,B 0,C 180,E1 -6023.49,E2 -6023.49} C_VEL
LIN {X 0,Y 495.706,Z 690.734,A -85,B 0,C 180,E1 -6025.936,E2 -6025.936} C_VEL
LIN {X 0,Y 495.978,Z 690.703,A -85,B 0,C 180,E1 -6027.565,E2 -6027.565} C_VEL
LIN {X 0,Y 495.975,Z 690.705,A -85,B 0,C 180,E1 -6030.001,E2 -6030.001} C_VEL
LIN {X 0,Y 495.977,Z 690.707,A -85,B 0,C 180,E1 -6032.438,E2 -6032.438} C_VEL
LIN {X 0,Y 495.855,Z 690.716,A -85,B 0,C 180,E1 -6035.695,E2 -6035.695} C_VEL
LIN {X 0,Y 495.814,Z 690.722,A -85,B 0,C 180,E1 -6038.15,E2 -6038.15} C_VEL
LIN {X 0,Y 495.816,Z 690.718,A -85,B 0,C 180,E1 -6041.447,E2 -6041.447} C_VEL
LIN {X 0,Y 495.783,Z 690.727,A -85,B 0,C 180,E1 -6044.784,E2 -6044.784} C_VEL
LIN {X 0,Y 495.778,Z 690.725,A -85,B 0,C 180,E1 -6048.236,E2 -6048.236} C_VEL
LIN {X 0,Y 495.742,Z 690.728,A -85,B 0,C 180,E1 -6051.63,E2 -6051.63} C_VEL
LIN {X 0,Y 495.708,Z 690.733,A -85,B 0,C 180,E1 -6054.278,E2 -6054.278} C_VEL
LIN {X 0,Y 495.723,Z 690.73,A -85,B 0,C 180,E1 -6056.981,E2 -6056.981} C_VEL
LIN {X 0,Y 495.7,Z 690.735,A -85,B 0,C 180,E1 -6059.752,E2 -6059.752} C_VEL
LIN {X 0,Y 495.73,Z 690.729,A -85,B 0,C 180,E1 -6062.598,E2 -6062.598} C_VEL
LIN {X 0,Y 495.719,Z 690.729,A -85,B 0,C 180,E1 -6065.541,E2 -6065.541} C_VEL
LIN {X 0,Y 495.728,Z 690.73,A -85,B 0,C 180,E1 -6068.762,E2 -6068.762} C_VEL
LIN {X 0,Y 495.704,Z 690.738,A -85,B 0,C 180,E1 -6071.788,E2 -6071.788} C_VEL
LIN {X 0,Y 495.738,Z 690.731,A -85,B 0,C 180,E1 -6075.142,E2 -6075.142} C_VEL
LIN {X 0,Y 495.706,Z 690.735,A -85,B 0,C 180,E1 -6078.213,E2 -6078.213} C_VEL
LIN {X 0,Y 495.71,Z 690.736,A -85,B 0,C 180,E1 -6081.404,E2 -6081.404} C_VEL
LIN {X 0,Y 495.717,Z 690.734,A -85,B 0,C 180,E1 -6084.459,E2 -6084.459} C_VEL
LIN {X 0,Y 495.73,Z 690.733,A -85,B 0,C 180,E1 -6087.403,E2 -6087.403} C_VEL
LIN {X 0,Y 495.702,Z 690.741,A -85,B 0,C 180,E1 -6090.249,E2 -6090.249} C_VEL
LIN {X 0,Y 495.761,Z 690.971,A -85,B 0,C 180,E1 -6091.422,E2 -6091.422} C_VEL
LIN {X 0,Y 496.052,Z 692.166,A -85,B 0,C 180,E1 -6091.548,E2 -6091.548} C_VEL
LIN {X 0,Y 498.417,Z 699.323,A -85,B 0,C 180,E1 -6091.738,E2 -6091.738} C_VEL
LIN {X 0,Y 497.928,Z 766.27,A -85,B 0,C 180,E1 -6092.753,E2 -6092.753} C_VEL
LIN {X 0,Y 497.8,Z 778.016,A -85,B 0,C 180,E1 -6093.063,E2 -6093.063} C_VEL
LIN {X 0,Y 497.609,Z 788.796,A -85,B 0,C 180,E1 -6093.47,E2 -6093.47} C_VEL
LIN {X 0,Y 497.415,Z 797.845,A -85,B 0,C 180,E1 -6093.911,E2 -6093.911} C_VEL
LIN {X 0,Y 497.135,Z 807.573,A -85,B 0,C 180,E1 -6094.502,E2 -6094.502} C_VEL
LIN {X 0,Y 496.842,Z 817.178,A -85,B 0,C 180,E1 -6095.225,E2 -6095.225} C_VEL
LIN {X 0,Y 496.509,Z 825.6,A -85,B 0,C 180,E1 -6095.986,E2 -6095.986} C_VEL
LIN {X 0,Y 496.298,Z 833.876,A -85,B 0,C 180,E1 -6096.89,E2 -6096.89} C_VEL
LIN {X 0,Y 496.077,Z 840.449,A -85,B 0,C 180,E1 -6097.73,E2 -6097.73} C_VEL
LIN {X 0,Y 495.751,Z 847.458,A -85,B 0,C 180,E1 -6098.807,E2 -6098.807} C_VEL
LIN {X 0,Y 495.631,Z 852.54,A -85,B 0,C 180,E1 -6099.735,E2 -6099.735} C_VEL
LIN {X 0,Y 495.467,Z 857.973,A -85,B 0,C 180,E1 -6100.959,E2 -6100.959} C_VEL
LIN {X 0,Y 495.341,Z 862.509,A -85,B 0,C 180,E1 -6102.285,E2 -6102.285} C_VEL
LIN {X 0,Y 495.197,Z 865.659,A -85,B 0,C 180,E1 -6103.51,E2 -6103.51} C_VEL
LIN {X 0,Y 495.165,Z 867.945,A -85,B 0,C 180,E1 -6104.83,E2 -6104.83} C_VEL
LIN {X 0,Y 495.142,Z 869.189,A -85,B 0,C 180,E1 -6106.037,E2 -6106.037} C_VEL
LIN {X 0,Y 495.158,Z 869.506,A -85,B 0,C 180,E1 -6106.874,E2 -6106.874} C_VEL
LIN {X 0,Y 495.213,Z 869.097,A -85,B 0,C 180,E1 -6108.308,E2 -6108.308} C_VEL
LIN {X 0,Y 495.234,Z 867.959,A -85,B 0,C 180,E1 -6109.369,E2 -6109.369} C_VEL
LIN {X 0,Y 495.291,Z 864.889,A -85,B 0,C 180,E1 -6111.02,E2 -6111.02} C_VEL
LIN {X 0,Y 495.428,Z 861.409,A -85,B 0,C 180,E1 -6112.255,E2 -6112.255} C_VEL
LIN {X 0,Y 495.568,Z 856.836,A -85,B 0,C 180,E1 -6113.485,E2 -6113.485} C_VEL
LIN {X 0,Y 495.708,Z 852.144,A -85,B 0,C 180,E1 -6114.508,E2 -6114.508} C_VEL
LIN {X 0,Y 495.942,Z 845.128,A -85,B 0,C 180,E1 -6115.733,E2 -6115.733} C_VEL
LIN {X 0,Y 496.181,Z 838.023,A -85,B 0,C 180,E1 -6116.752,E2 -6116.752} C_VEL
LIN {X 0,Y 496.442,Z 831.31,A -85,B 0,C 180,E1 -6117.566,E2 -6117.566} C_VEL
LIN {X 0,Y 496.745,Z 822.216,A -85,B 0,C 180,E1 -6118.48,E2 -6118.48} C_VEL
LIN {X 0,Y 497.022,Z 813.727,A -85,B 0,C 180,E1 -6119.19,E2 -6119.19} C_VEL
LIN {X 0,Y 497.29,Z 805.004,A -85,B 0,C 180,E1 -6119.797,E2 -6119.797} C_VEL
LIN {X 0,Y 497.534,Z 794.05,A -85,B 0,C 180,E1 -6120.405,E2 -6120.405} C_VEL
LIN {X 0,Y 497.775,Z 783.314,A -85,B 0,C 180,E1 -6120.859,E2 -6120.859} C_VEL
LIN {X 0,Y 497.851,Z 772.805,A -85,B 0,C 180,E1 -6121.188,E2 -6121.188} C_VEL
LIN {X 0,Y 498.026,Z 760.252,A -85,B 0,C 180,E1 -6121.44,E2 -6121.44} C_VEL
LIN {X 0,Y 498.319,Z 698.291,A -85,B 0,C 180,E1 -6122.374,E2 -6122.374} C_VEL
LIN {X 0,Y 496.152,Z 691.726,A -85,B 0,C 180,E1 -6122.562,E2 -6122.562} C_VEL
LIN {X 0,Y 495.973,Z 690.871,A -85,B 0,C 180,E1 -6122.69,E2 -6122.69} C_VEL
LIN {X 0,Y 495.887,Z 690.717,A -85,B 0,C 180,E1 -6125.693,E2 -6125.693} C_VEL
LIN {X 0,Y 495.84,Z 690.719,A -85,B 0,C 180,E1 -6128.97,E2 -6128.97} C_VEL
LIN {X 0,Y 495.836,Z 690.722,A -85,B 0,C 180,E1 -6132.034,E2 -6132.034} C_VEL
LIN {X 0,Y 495.831,Z 690.719,A -85,B 0,C 180,E1 -6135.451,E2 -6135.451} C_VEL
LIN {X 0,Y 495.785,Z 690.729,A -85,B 0,C 180,E1 -6138.237,E2 -6138.237} C_VEL
LIN {X 0,Y 495.781,Z 690.73,A -85,B 0,C 180,E1 -6140.756,E2 -6140.756} C_VEL
LIN {X 0,Y 495.753,Z 690.728,A -85,B 0,C 180,E1 -6143.387,E2 -6143.387} C_VEL
LIN {X 0,Y 495.766,Z 690.727,A -85,B 0,C 180,E1 -6146.069,E2 -6146.069} C_VEL
LIN {X 0,Y 495.751,Z 690.735,A -85,B 0,C 180,E1 -6148.816,E2 -6148.816} C_VEL
LIN {X 0,Y 495.761,Z 690.727,A -85,B 0,C 180,E1 -6151.725,E2 -6151.725} C_VEL
LIN {X 0,Y 495.769,Z 690.73,A -85,B 0,C 180,E1 -6154.692,E2 -6154.692} C_VEL
LIN {X 0,Y 495.735,Z 690.733,A -85,B 0,C 180,E1 -6157.561,E2 -6157.561} C_VEL
LIN {X 0,Y 495.773,Z 690.728,A -85,B 0,C 180,E1 -6160.699,E2 -6160.699} C_VEL
LIN {X 0,Y 495.734,Z 690.731,A -85,B 0,C 180,E1 -6164.001,E2 -6164.001} C_VEL
LIN {X 0,Y 495.731,Z 690.736,A -85,B 0,C 180,E1 -6167.116,E2 -6167.116} C_VEL
LIN {X 0,Y 495.76,Z 690.729,A -85,B 0,C 180,E1 -6169.953,E2 -6169.953} C_VEL
LIN {X 0,Y 495.724,Z 690.731,A -85,B 0,C 180,E1 -6172.554,E2 -6172.554} C_VEL
LIN {X 0,Y 495.776,Z 690.732,A -85,B 0,C 180,E1 -6175.455,E2 -6175.455} C_VEL
LIN {X 0,Y 495.761,Z 690.732,A -85,B 0,C 180,E1 -6178.363,E2 -6178.363} C_VEL
LIN {X 0,Y 495.829,Z 690.916,A -85,B 0,C 180,E1 -6180.289,E2 -6180.289} C_VEL
LIN {X 0,Y 499.486,Z 707.298,A -85,B 0,C 180,E1 -6182.634,E2 -6182.634} C_VEL
LIN {X 0,Y 498.585,Z 731.096,A -85,B 0,C 180,E1 -6185.649,E2 -6185.649} C_VEL
LIN {X 0,Y 497.921,Z 753.685,A -85,B 0,C 180,E1 -6188.469,E2 -6188.469} C_VEL
LIN {X 0,Y 497.191,Z 779.03,A -85,B 0,C 180,E1 -6191.558,E2 -6191.558} C_VEL
LIN {X 0,Y 496.69,Z 798.526,A -85,B 0,C 180,E1 -6193.924,E2 -6193.924} C_VEL
LIN {X 0,Y 498.096,Z 810.55,A -85,B 0,C 180,E1 -6194.172,E2 -6194.172} C_VEL
LIN {X 0,Y 498.473,Z 817.097,A -85,B 0,C 180,E1 -6194.28,E2 -6194.28} C_VEL
LIN {X 0,Y 497.988,Z 908.908,A -85,B 0,C 180,E1 -6195.622,E2 -6195.622} C_VEL
LIN {X 0,Y 497.619,Z 922.342,A -85,B 0,C 180,E1 -6195.976,E2 -6195.976} C_VEL
LIN {X 0,Y 497.294,Z 935.79,A -85,B 0,C 180,E1 -6196.514,E2 -6196.514} C_VEL
LIN {X 0,Y 496.927,Z 948.147,A -85,B 0,C 180,E1 -6197.196,E2 -6197.196} C_VEL
LIN {X 0,Y 496.567,Z 960.185,A -85,B 0,C 180,E1 -6198.053,E2 -6198.053} C_VEL
LIN {X 0,Y 496.159,Z 970.55,A -85,B 0,C 180,E1 -6198.975,E2 -6198.975} C_VEL
LIN {X 0,Y 495.856,Z 979.9,A -85,B 0,C 180,E1 -6200,E2 -6200} C_VEL
LIN {X 0,Y 495.544,Z 989.02,A -85,B 0,C 180,E1 -6201.229,E2 -6201.229} C_VEL
LIN {X 0,Y 495.314,Z 996.377,A -85,B 0,C 180,E1 -6202.457,E2 -6202.457} C_VEL
LIN {X 0,Y 495.205,Z 1002.375,A -85,B 0,C 180,E1 -6203.71,E2 -6203.71} C_VEL
LIN {X 0,Y 495.152,Z 1006.207,A -85,B 0,C 180,E1 -6204.705,E2 -6204.705} C_VEL
LIN {X 0,Y 495.089,Z 1009.913,A -85,B 0,C 180,E1 -6205.929,E2 -6205.929} C_VEL
LIN {X 0,Y 495.074,Z 1011.827,A -85,B 0,C 180,E1 -6206.744,E2 -6206.744} C_VEL
LIN {X 0,Y 495.015,Z 1013.257,A -85,B 0,C 180,E1 -6207.558,E2 -6207.558} C_VEL
LIN {X 0,Y 494.985,Z 1014.279,A -85,B 0,C 180,E1 -6208.372,E2 -6208.372} C_VEL
LIN {X 0,Y 494.943,Z 1014.899,A -85,B 0,C 180,E1 -6209.185,E2 -6209.185} C_VEL
LIN {X 0,Y 494.933,Z 1015.119,A -85,B 0,C 180,E1 -6209.999,E2 -6209.999} C_VEL
LIN {X 0,Y 494.943,Z 1014.898,A -85,B 0,C 180,E1 -6210.812,E2 -6210.812} C_VEL
LIN {X 0,Y 494.986,Z 1014.278,A -85,B 0,C 180,E1 -6211.626,E2 -6211.626} C_VEL
LIN {X 0,Y 495.015,Z 1013.256,A -85,B 0,C 180,E1 -6212.44,E2 -6212.44} C_VEL
LIN {X 0,Y 495.074,Z 1011.824,A -85,B 0,C 180,E1 -6213.254,E2 -6213.254} C_VEL
LIN {X 0,Y 495.07,Z 1008.798,A -85,B 0,C 180,E1 -6214.477,E2 -6214.477} C_VEL
LIN {X 0,Y 495.196,Z 1004.723,A -85,B 0,C 180,E1 -6215.7,E2 -6215.7} C_VEL
LIN {X 0,Y 495.27,Z 998.544,A -85,B 0,C 180,E1 -6217.111,E2 -6217.111} C_VEL
LIN {X 0,Y 495.458,Z 991.6,A -85,B 0,C 180,E1 -6218.359,E2 -6218.359} C_VEL
LIN {X 0,Y 495.725,Z 983.128,A -85,B 0,C 180,E1 -6219.588,E2 -6219.588} C_VEL
LIN {X 0,Y 495.986,Z 974.453,A -85,B 0,C 180,E1 -6220.614,E2 -6220.614} C_VEL
LIN {X 0,Y 496.398,Z 963.775,A -85,B 0,C 180,E1 -6221.638,E2 -6221.638} C_VEL
LIN {X 0,Y 496.806,Z 951.916,A -85,B 0,C 180,E1 -6222.551,E2 -6222.551} C_VEL
LIN {X 0,Y 497.119,Z 939.724,A -85,B 0,C 180,E1 -6223.28,E2 -6223.28} C_VEL
LIN {X 0,Y 497.558,Z 927.245,A -85,B 0,C 180,E1 -6223.84,E2 -6223.84} C_VEL
LIN {X 0,Y 497.834,Z 914.439,A -85,B 0,C 180,E1 -6224.25,E2 -6224.25} C_VEL
LIN {X 0,Y 498.014,Z 899.259,A -85,B 0,C 180,E1 -6224.531,E2 -6224.531} C_VEL
LIN {X 0,Y 498.441,Z 813.301,A -85,B 0,C 180,E1 -6225.772,E2 -6225.772} C_VEL
LIN {X 0,Y 496.668,Z 798.263,A -85,B 0,C 180,E1 -6226.073,E2 -6226.073} C_VEL
LIN {X 0,Y 497.239,Z 774.286,A -85,B 0,C 180,E1 -6228.969,E2 -6228.969} C_VEL
LIN {X 0,Y 497.953,Z 749.71,A -85,B 0,C 180,E1 -6231.962,E2 -6231.962} C_VEL
LIN {X 0,Y 498.812,Z 722.529,A -85,B 0,C 180,E1 -6235.346,E2 -6235.346} C_VEL
LIN {X 0,Y 499.336,Z 706.758,A -85,B 0,C 180,E1 -6237.344,E2 -6237.344} C_VEL
LIN {X 0,Y 495.808,Z 690.891,A -85,B 0,C 180,E1 -6239.61,E2 -6239.61} C_VEL
LIN {X 0,Y 495.762,Z 690.734,A -85,B 0,C 180,E1 -6242.593,E2 -6242.593} C_VEL
LIN {X 0,Y 495.742,Z 690.731,A -85,B 0,C 180,E1 -6245.536,E2 -6245.536} C_VEL
LIN {X 0,Y 495.756,Z 690.734,A -85,B 0,C 180,E1 -6248.767,E2 -6248.767} C_VEL
LIN {X 0,Y 495.749,Z 690.729,A -85,B 0,C 180,E1 -6251.78,E2 -6251.78} C_VEL
LIN {X 0,Y 495.742,Z 690.731,A -85,B 0,C 180,E1 -6255.138,E2 -6255.138} C_VEL
LIN {X 0,Y 495.769,Z 690.727,A -85,B 0,C 180,E1 -6258.22,E2 -6258.22} C_VEL
LIN {X 0,Y 495.743,Z 690.732,A -85,B 0,C 180,E1 -6261.408,E2 -6261.408} C_VEL
LIN {X 0,Y 495.748,Z 690.725,A -85,B 0,C 180,E1 -6264.462,E2 -6264.462} C_VEL
LIN {X 0,Y 495.758,Z 690.732,A -85,B 0,C 180,E1 -6267.405,E2 -6267.405} C_VEL
LIN {X 0,Y 495.771,Z 690.725,A -85,B 0,C 180,E1 -6270.254,E2 -6270.254} C_VEL
LIN {X 0,Y 495.823,Z 690.724,A -85,B 0,C 180,E1 -6273.248,E2 -6273.248} C_VEL
LIN {X 0,Y 495.742,Z 690.734,A -85,B 0,C 180,E1 -6275.724,E2 -6275.724} C_VEL
LIN {X 0,Y 495.736,Z 690.727,A -85,B 0,C 180,E1 -6278.371,E2 -6278.371} C_VEL
LIN {X 0,Y 495.773,Z 690.725,A -85,B 0,C 180,E1 -6280.971,E2 -6280.971} C_VEL
LIN {X 0,Y 495.767,Z 690.728,A -85,B 0,C 180,E1 -6283.53,E2 -6283.53} C_VEL
LIN {X 0,Y 495.782,Z 690.726,A -85,B 0,C 180,E1 -6286.055,E2 -6286.055} C_VEL
LIN {X 0,Y 495.839,Z 690.718,A -85,B 0,C 180,E1 -6288.555,E2 -6288.555} C_VEL
LIN {X 0,Y 495.861,Z 690.715,A -85,B 0,C 180,E1 -6291.852,E2 -6291.852} C_VEL
LIN {X 0,Y 495.878,Z 690.716,A -85,B 0,C 180,E1 -6294.306,E2 -6294.306} C_VEL
LIN {X 0,Y 495.98,Z 690.699,A -85,B 0,C 180,E1 -6297.564,E2 -6297.564} C_VEL
LIN {X 0,Y 495.984,Z 690.701,A -85,B 0,C 180,E1 -6300,E2 -6300} C_VEL
LIN {X 0,Y 495.98,Z 690.707,A -85,B 0,C 180,E1 -6302.437,E2 -6302.437} C_VEL
LIN {X 0,Y 495.878,Z 690.71,A -85,B 0,C 180,E1 -6305.694,E2 -6305.694} C_VEL
LIN {X 0,Y 495.861,Z 690.715,A -85,B 0,C 180,E1 -6308.148,E2 -6308.148} C_VEL
LIN {X 0,Y 495.843,Z 690.715,A -85,B 0,C 180,E1 -6311.446,E2 -6311.446} C_VEL
LIN {X 0,Y 495.778,Z 690.732,A -85,B 0,C 180,E1 -6314.783,E2 -6314.783} C_VEL
LIN {X 0,Y 495.753,Z 690.731,A -85,B 0,C 180,E1 -6317.32,E2 -6317.32} C_VEL
LIN {X 0,Y 495.76,Z 690.726,A -85,B 0,C 180,E1 -6319.891,E2 -6319.891} C_VEL
LIN {X 0,Y 495.747,Z 690.731,A -85,B 0,C 180,E1 -6322.861,E2 -6322.861} C_VEL
LIN {X 0,Y 495.749,Z 690.729,A -85,B 0,C 180,E1 -6326.071,E2 -6326.071} C_VEL
LIN {X 0,Y 495.759,Z 690.723,A -85,B 0,C 180,E1 -6328.816,E2 -6328.816} C_VEL
LIN {X 0,Y 495.747,Z 690.731,A -85,B 0,C 180,E1 -6331.727,E2 -6331.727} C_VEL
LIN {X 0,Y 495.765,Z 690.726,A -85,B 0,C 180,E1 -6334.696,E2 -6334.696} C_VEL
LIN {X 0,Y 495.723,Z 690.738,A -85,B 0,C 180,E1 -6337.563,E2 -6337.563} C_VEL
LIN {X 0,Y 495.759,Z 690.727,A -85,B 0,C 180,E1 -6340.701,E2 -6340.701} C_VEL
LIN {X 0,Y 495.721,Z 690.739,A -85,B 0,C 180,E1 -6344.003,E2 -6344.003} C_VEL
LIN {X 0,Y 495.71,Z 690.732,A -85,B 0,C 180,E1 -6347.117,E2 -6347.117} C_VEL
LIN {X 0,Y 495.787,Z 690.894,A -85,B 0,C 180,E1 -6349.275,E2 -6349.275} C_VEL
LIN {X 0,Y 495.977,Z 691.825,A -85,B 0,C 180,E1 -6349.408,E2 -6349.408} C_VEL
LIN {X 0,Y 498.697,Z 699.343,A -85,B 0,C 180,E1 -6349.626,E2 -6349.626} C_VEL
LIN {X 0,Y 498.285,Z 771.437,A -85,B 0,C 180,E1 -6350.703,E2 -6350.703} C_VEL
LIN {X 0,Y 498.24,Z 778.469,A -85,B 0,C 180,E1 -6350.878,E2 -6350.878} C_VEL
LIN {X 0,Y 497.541,Z 784.256,A -85,B 0,C 180,E1 -6351.035,E2 -6351.035} C_VEL
LIN {X 0,Y 494.632,Z 793.507,A -85,B 0,C 180,E1 -6351.3,E2 -6351.3} C_VEL
LIN {X 0,Y 491.702,Z 802.467,A -85,B 0,C 180,E1 -6351.646,E2 -6351.646} C_VEL
LIN {X 0,Y 490.972,Z 807.684,A -85,B 0,C 180,E1 -6351.928,E2 -6351.928} C_VEL
LIN {X 0,Y 490.647,Z 819.479,A -85,B 0,C 180,E1 -6352.76,E2 -6352.76} C_VEL
LIN {X 0,Y 490.286,Z 829.972,A -85,B 0,C 180,E1 -6353.699,E2 -6353.699} C_VEL
LIN {X 0,Y 489.887,Z 839.265,A -85,B 0,C 180,E1 -6354.724,E2 -6354.724} C_VEL
LIN {X 0,Y 489.475,Z 848.179,A -85,B 0,C 180,E1 -6355.948,E2 -6355.948} C_VEL
LIN {X 0,Y 489.205,Z 855.253,A -85,B 0,C 180,E1 -6357.16,E2 -6357.16} C_VEL
LIN {X 0,Y 488.93,Z 861.122,A -85,B 0,C 180,E1 -6358.409,E2 -6358.409} C_VEL
LIN {X 0,Y 488.718,Z 866.155,A -85,B 0,C 180,E1 -6359.782,E2 -6359.782} C_VEL
LIN {X 0,Y 488.557,Z 870.253,A -85,B 0,C 180,E1 -6361.343,E2 -6361.343} C_VEL
LIN {X 0,Y 488.464,Z 873.122,A -85,B 0,C 180,E1 -6363.133,E2 -6363.133} C_VEL
LIN {X 0,Y 488.387,Z 874.033,A -85,B 0,C 180,E1 -6364.426,E2 -6364.426} C_VEL
LIN {X 0,Y 488.399,Z 874.073,A -85,B 0,C 180,E1 -6365.337,E2 -6365.337} C_VEL
LIN {X 0,Y 488.375,Z 873.688,A -85,B 0,C 180,E1 -6366.24,E2 -6366.24} C_VEL
LIN {X 0,Y 488.416,Z 872.831,A -85,B 0,C 180,E1 -6367.14,E2 -6367.14} C_VEL
LIN {X 0,Y 488.476,Z 871.494,A -85,B 0,C 180,E1 -6368.034,E2 -6368.034} C_VEL
LIN {X 0,Y 488.619,Z 869.003,A -85,B 0,C 180,E1 -6369.217,E2 -6369.217} C_VEL
LIN {X 0,Y 488.781,Z 864.649,A -85,B 0,C 180,E1 -6370.69,E2 -6370.69} C_VEL
LIN {X 0,Y 488.99,Z 859.469,A -85,B 0,C 180,E1 -6372.002,E2 -6372.002} C_VEL
LIN {X 0,Y 489.216,Z 852.911,A -85,B 0,C 180,E1 -6373.304,E2 -6373.304} C_VEL
LIN {X 0,Y 489.604,Z 844.526,A -85,B 0,C 180,E1 -6374.619,E2 -6374.619} C_VEL
LIN {X 0,Y 489.909,Z 836.234,A -85,B 0,C 180,E1 -6375.674,E2 -6375.674} C_VEL
LIN {X 0,Y 490.282,Z 826.996,A -85,B 0,C 180,E1 -6376.637,E2 -6376.637} C_VEL
LIN {X 0,Y 490.616,Z 817.069,A -85,B 0,C 180,E1 -6377.477,E2 -6377.477} C_VEL
LIN {X 0,Y 490.944,Z 805.936,A -85,B 0,C 180,E1 -6378.231,E2 -6378.231} C_VEL
LIN {X 0,Y 491.177,Z 793.852,A -85,B 0,C 180,E1 -6378.864,E2 -6378.864} C_VEL
LIN {X 0,Y 491.354,Z 781.36,A -85,B 0,C 180,E1 -6379.337,E2 -6379.337} C_VEL
LIN {X 0,Y 491.403,Z 768.499,A -85,B 0,C 180,E1 -6379.651,E2 -6379.651} C_VEL
LIN {X 0,Y 491.83,Z 700.789,A -85,B 0,C 180,E1 -6380.657,E2 -6380.657} C_VEL
